KUKA KRL program: MyProgram_339().src

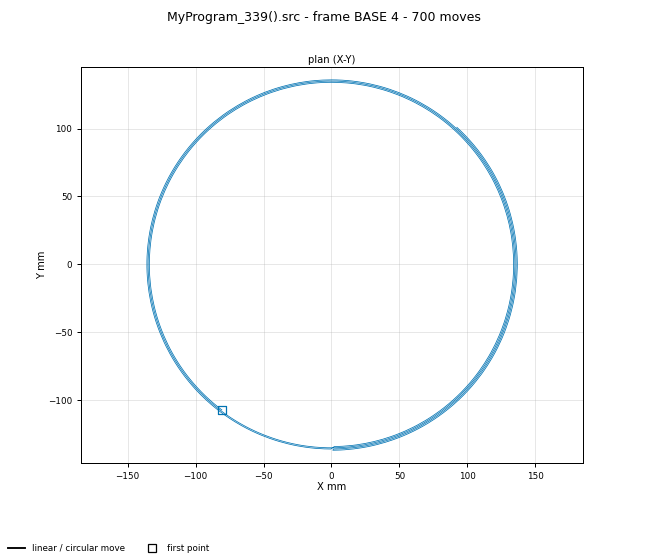
[picture p0: tool path of MyProgram_339().src in frame BASE 4, 700 of 700 moves have a stored position in this frame; points joined in program order, loops and branches not executed]
&ACCESS RVP
&REL 1
&PARAM TEMPLATE = C:\KRC\Roboter\Template\vorgabe
&PARAM EDITMASK = *
DEF MyProgram_339()
; ---- Setting reference (Base) ----
$BASE = BASE_DATA[4]

; --------------------------
; ---- Setting tool (TCP) ----
$TOOL = TOOL_DATA[3]
; --------------------------

$VEL.CP = VEL_APROX_PRINT
Startdeposition()
$VEL.CP = VEL_PRINT
LIN {X -80.6582,Y -106.9926,Z 191,A -116.6087,B 1.012,C 0.191,E1 0.9414,E2 209.5194} C_DIS
LIN {X -83.2208,Y -105.0121,Z 191,A -118.2945,B 1.0123,C 0.1893,E1 0.9375,E2 211.2466} C_DIS
LIN {X -86.7658,Y -102.1022,Z 191,A -120.2784,B 1.0128,C 0.1864,E1 0.9332,E2 213.2337} C_DIS
LIN {X -89.4407,Y -99.7673,Z 191,A -122.0496,B 1.0132,C 0.1842,E1 0.9294,E2 215.0396} C_DIS
LIN {X -92.5437,Y -96.8959,Z 191,A -124.0147,B 1.0137,C 0.1814,E1 0.9254,E2 217.0261} C_DIS
LIN {X -95.7328,Y -93.7464,Z 191,A -126.0613,B 1.0143,C 0.1781,E1 0.9213,E2 219.0903} C_DIS
LIN {X -98.7291,Y -90.5855,Z 191,A -128.1724,B 1.0149,C 0.1749,E1 0.9171,E2 221.2352} C_DIS
LIN {X -101.4585,Y -87.5176,Z 191,A -129.9716,B 1.0154,C 0.1717,E1 0.9138,E2 223.04} C_DIS
LIN {X -103.9869,Y -84.4986,Z 191,A -131.8725,B 1.0159,C 0.1685,E1 0.9103,E2 224.97} C_DIS
LIN {X -106.5269,Y -81.2724,Z 191,A -133.8231,B 1.0165,C 0.165,E1 0.9069,E2 226.9467} C_DIS
LIN {X -108.5873,Y -78.4983,Z 191,A -135.5077,B 1.017,C 0.162,E1 0.9041,E2 228.6589} C_DIS
LIN {X -111.0789,Y -74.9311,Z 191,A -137.5649,B 1.0176,C 0.158,E1 0.9008,E2 230.7422} C_DIS
LIN {X -113.2039,Y -71.6803,Z 191,A -139.4925,B 1.0182,C 0.1544,E1 0.8978,E2 232.7051} C_DIS
LIN {X -115.4642,Y -67.9793,Z 191,A -141.5321,B 1.0188,C 0.1502,E1 0.8948,E2 234.769} C_DIS
LIN {X -117.2157,Y -64.9126,Z 191,A -143.1833,B 1.0193,C 0.1467,E1 0.8925,E2 236.4385} C_DIS
LIN {X -118.7707,Y -62.0179,Z 191,A -144.823,B 1.0198,C 0.1433,E1 0.8903,E2 238.1089} C_DIS
LIN {X -120.4109,Y -58.7718,Z 191,A -146.5306,B 1.0203,C 0.1396,E1 0.8882,E2 239.8362} C_DIS
LIN {X -121.8201,Y -55.7917,Z 191,A -148.1544,B 1.0208,C 0.1361,E1 0.8862,E2 241.4877} C_DIS
LIN {X -123.1512,Y -52.788,Z 191,A -149.9155,B 1.0213,C 0.1325,E1 0.8842,E2 243.2951} C_DIS
LIN {X -124.8857,Y -48.5406,Z 191,A -151.9995,B 1.0219,C 0.1275,E1 0.882,E2 245.3943} C_DIS
LIN {X -126.0829,Y -45.3403,Z 191,A -153.6668,B 1.0224,C 0.1236,E1 0.8804,E2 247.088} C_DIS
LIN {X -127.2363,Y -41.9963,Z 191,A -155.4129,B 1.0228,C 0.1196,E1 0.8788,E2 248.8638} C_DIS
LIN {X -128.2213,Y -38.8855,Z 191,A -156.9641,B 1.0233,C 0.1159,E1 0.8775,E2 250.4347} C_DIS
LIN {X -129.2898,Y -35.1747,Z 191,A -159.129,B 1.0238,C 0.1112,E1 0.8758,E2 252.6651} C_DIS
LIN {X -130.2828,Y -31.2902,Z 191,A -160.9064,B 1.0243,C 0.1065,E1 0.8746,E2 254.4498} C_DIS
LIN {X -131.0111,Y -28.086,Z 191,A -162.5308,B 1.0247,C 0.1026,E1 0.8736,E2 256.1016} C_DIS
LIN {X -131.6609,Y -24.8637,Z 191,A -164.1583,B 1.0251,C 0.0986,E1 0.8727,E2 257.7568} C_DIS
LIN {X -132.289,Y -21.2821,Z 191,A -165.9785,B 1.0255,C 0.0941,E1 0.8719,E2 259.61} C_DIS
LIN {X -132.7236,Y -18.3714,Z 191,A -167.4143,B 1.0258,C 0.0905,E1 0.8713,E2 261.0676} C_DIS
LIN {X -133.1719,Y -14.7703,Z 191,A -169.1065,B 1.0262,C 0.0861,E1 0.8707,E2 262.7767} C_DIS
LIN {X -133.4937,Y -11.4993,Z 191,A -170.8721,B 1.0266,C 0.0819,E1 0.8702,E2 264.5869} C_DIS
LIN {X -133.7359,Y -8.2135,Z 191,A -172.4215,B 1.0269,C 0.0779,E1 0.8699,E2 266.1531} C_DIS
LIN {X -133.8842,Y -5.2709,Z 191,A -173.969,B 1.0271,C 0.0741,E1 0.8697,E2 267.7357} C_DIS
LIN {X -133.9734,Y -1.9867,Z 191,A -175.5899,B 1.0274,C 0.07,E1 0.8697,E2 269.3826} C_DIS
LIN {X -133.9855,Y 0.9522,Z 191,A -177.2293,B 1.0277,C 0.0661,E1 0.8697,E2 271.0686} C_DIS
LIN {X -133.8989,Y 4.8936,Z 191,A -179.0532,B 1.028,C 0.0613,E1 0.8698,E2 272.9085} C_DIS
LIN {X -133.7428,Y 8.102,Z 191,A 179.4246,B 1.0282,C 0.0573,E1 0.87,E2 274.4481} C_DIS
LIN {X -133.5228,Y 11.1541,Z 191,A 177.8434,B 1.0284,C 0.0534,E1 0.8704,E2 276.0618} C_DIS
LIN {X -133.1725,Y 14.7653,Z 191,A 176.0918,B 1.0287,C 0.0489,E1 0.8709,E2 277.8368} C_DIS
LIN {X -132.8155,Y 17.6872,Z 191,A 174.5479,B 1.0288,C 0.0452,E1 0.8714,E2 279.4144} C_DIS
LIN {X -132.3404,Y 20.951,Z 191,A 172.9492,B 1.029,C 0.0411,E1 0.8721,E2 281.035} C_DIS
LIN {X -131.7256,Y 24.525,Z 191,A 171.1308,B 1.0292,C 0.0366,E1 0.873,E2 282.8846} C_DIS
LIN {X -131.0843,Y 27.747,Z 191,A 169.5917,B 1.0292,C 0.0327,E1 0.8739,E2 284.4389} C_DIS
LIN {X -130.4904,Y 30.4188,Z 191,A 167.994,B 1.0294,C 0.0291,E1 0.8749,E2 286.0866} C_DIS
LIN {X -129.5576,Y 34.1706,Z 191,A 166.4075,B 1.0295,C 0.0248,E1 0.876,E2 287.6642} C_DIS
LIN {X -128.6838,Y 37.3263,Z 191,A 164.6242,B 1.0296,C 0.0207,E1 0.8774,E2 289.4919} C_DIS
LIN {X -127.832,Y 40.1504,Z 191,A 163.1708,B 1.0296,C 0.0172,E1 0.8786,E2 290.967} C_DIS
LIN {X -126.699,Y 43.5904,Z 191,A 161.2988,B 1.0297,C 0.0129,E1 0.8803,E2 292.8757} C_DIS
LIN {X -125.2326,Y 47.6435,Z 191,A 159.0965,B 1.0297,C 0.0079,E1 0.8825,E2 295.1186} C_DIS
LIN {X -123.7899,Y 51.2722,Z 191,A 157.5034,B 1.0298,C 0.0038,E1 0.8842,E2 296.7016} C_DIS
LIN {X -122.6365,Y 53.9772,Z 191,A 155.7935,B 1.0298,C 0.0003,E1 0.8861,E2 298.463} C_DIS
LIN {X -121.3505,Y 56.8073,Z 191,A 154.4119,B 1.0298,C -0.003,E1 0.8878,E2 299.8497} C_DIS
LIN {X -119.8894,Y 59.8292,Z 191,A 152.7456,B 1.0298,C -0.0066,E1 0.8898,E2 301.5415} C_DIS
LIN {X -118.166,Y 63.1666,Z 191,A 150.9408,B 1.0298,C -0.0105,E1 0.8922,E2 303.3678} C_DIS
LIN {X -116.5834,Y 66.0427,Z 191,A 149.3435,B 1.0298,C -0.0139,E1 0.8944,E2 304.9862} C_DIS
LIN {X -114.7495,Y 69.1791,Z 191,A 147.4569,B 1.0297,C -0.0176,E1 0.8972,E2 306.9092} C_DIS
LIN {X -112.5008,Y 72.779,Z 191,A 145.4626,B 1.0296,C -0.0217,E1 0.9002,E2 308.9225} C_DIS
LIN {X -110.4885,Y 75.7988,Z 191,A 143.804,B 1.0296,C -0.0251,E1 0.9028,E2 310.592} C_DIS
LIN {X -108.7858,Y 78.2236,Z 191,A 142.3734,B 1.0294,C -0.0279,E1 0.9052,E2 312.0401} C_DIS
LIN {X -106.837,Y 80.8644,Z 191,A 140.9363,B 1.0294,C -0.0308,E1 0.9076,E2 313.48} C_DIS
LIN {X -105.0171,Y 83.2145,Z 191,A 139.2547,B 1.0293,C -0.0334,E1 0.9106,E2 315.2063} C_DIS
LIN {X -102.22,Y 86.6272,Z 191,A 137.1876,B 1.0291,C -0.0372,E1 0.9144,E2 317.2919} C_DIS
LIN {X -99.2737,Y 89.9882,Z 191,A 135.0621,B 1.0291,C -0.0408,E1 0.9184,E2 319.4397} C_DIS
LIN {X -96.4718,Y 92.9862,Z 191,A 133.1168,B 1.0289,C -0.0439,E1 0.9222,E2 321.4046} C_DIS
LIN {X -93.5796,Y 95.8964,Z 191,A 131.3002,B 1.0287,C -0.047,E1 0.9258,E2 323.2269} C_DIS
LIN {X -90.5814,Y 98.7329,Z 191,A 129.2709,B 1.0287,C -0.0498,E1 0.93,E2 325.2836} C_DIS
LIN {X -87.5151,Y 101.4607,Z 191,A 127.5032,B 1.0285,C -0.0526,E1 0.9338,E2 327.0516} C_DIS
LIN {X -84.499,Y 103.9866,Z 191,A 125.6464,B 1.0283,C -0.0551,E1 0.9379,E2 328.9262} C_DIS
LIN {X -81.2745,Y 106.5253,Z 191,A 123.7533,B 1.0283,C -0.0575,E1 0.9421,E2 330.8331} C_DIS
LIN {X -78.9345,Y 108.2711,Z 191,A 122.3198,B 1.0281,C -0.0591,E1 0.9454,E2 332.2857} C_DIS
LIN {X -76.0804,Y 110.2952,Z 191,A 120.8532,B 1.0281,C -0.0611,E1 0.9488,E2 333.7483} C_DIS
LIN {X -73.3552,Y 112.1263,Z 191,A 119.2639,B 1.0279,C -0.0627,E1 0.9526,E2 335.3564} C_DIS
LIN {X -70.57,Y 113.8995,Z 191,A 117.9357,B 1.0279,C -0.0644,E1 0.9557,E2 336.6749} C_DIS
LIN {X -67.7643,Y 115.5905,Z 191,A 116.367,B 1.0277,C -0.0658,E1 0.9596,E2 338.2606} C_DIS
LIN {X -64.918,Y 117.2127,Z 191,A 114.8879,B 1.0277,C -0.0671,E1 0.9632,E2 339.7473} C_DIS
LIN {X -62.0091,Y 118.7753,Z 191,A 113.3972,B 1.0275,C -0.0684,E1 0.967,E2 341.2454} C_DIS
LIN {X -58.7582,Y 120.4177,Z 191,A 111.7712,B 1.0275,C -0.0697,E1 0.9711,E2 342.8778} C_DIS
LIN {X -55.7891,Y 121.8213,Z 191,A 110.3091,B 1.0274,C -0.0708,E1 0.9748,E2 344.3452} C_DIS
LIN {X -52.7868,Y 123.1518,Z 191,A 108.852,B 1.0274,C -0.0718,E1 0.9786,E2 345.8071} C_DIS
LIN {X -50.0675,Y 124.2814,Z 191,A 107.5514,B 1.0273,C -0.0726,E1 0.982,E2 347.1114} C_DIS
LIN {X -47.007,Y 125.471,Z 191,A 106.1033,B 1.0273,C -0.0733,E1 0.9859,E2 348.5633} C_DIS
LIN {X -43.9186,Y 126.5851,Z 191,A 104.6605,B 1.0272,C -0.074,E1 0.9897,E2 350.0095} C_DIS
LIN {X -40.4653,Y 127.7314,Z 191,A 103.0676,B 1.0272,C -0.0747,E1 0.994,E2 351.6055} C_DIS
LIN {X -37.7794,Y 128.5511,Z 191,A 101.8102,B 1.0271,C -0.0751,E1 0.9974,E2 352.8683} C_DIS
LIN {X -34.4694,Y 129.4779,Z 191,A 100.3485,B 1.0271,C -0.0756,E1 1.0014,E2 354.3284} C_DIS
LIN {X -31.2848,Y 130.2841,Z 191,A 98.9263,B 1.0271,C -0.0759,E1 1.0053,E2 355.7517} C_DIS
LIN {X -28.0812,Y 131.0121,Z 191,A 97.51,B 1.027,C -0.0761,E1 1.0092,E2 357.1686} C_DIS
LIN {X -24.8607,Y 131.6614,Z 191,A 96.0961,B 1.027,C -0.0763,E1 1.0131,E2 358.5827} C_DIS
LIN {X -21.2683,Y 132.2912,Z 191,A 94.5183,B 1.027,C -0.0763,E1 1.0175,E2 360.1619} C_DIS
LIN {X -18.3553,Y 132.7259,Z 191,A 93.2012,B 1.027,C -0.0762,E1 1.0212,E2 361.4844} C_DIS
LIN {X -14.7645,Y 133.1725,Z 191,A 91.7254,B 1.027,C -0.0762,E1 1.0254,E2 362.9521} C_DIS
LIN {X -10.5648,Y 133.5726,Z 191,A 89.7687,B 1.027,C -0.0755,E1 1.0309,E2 364.9241} C_DIS
LIN {X -6.9098,Y 133.8097,Z 191,A 88.3975,B 1.027,C -0.0755,E1 1.0347,E2 366.2741} C_DIS
LIN {X -3.616,Y 133.9392,Z 191,A 87.0209,B 1.027,C -0.0751,E1 1.0386,E2 367.6467} C_DIS
LIN {X 0.006,Y 133.99,Z 191,A 85.3856,B 1.0271,C -0.0743,E1 1.0433,E2 369.2905} C_DIS
LIN {X 4.3014,Y 133.9201,Z 191,A 83.5553,B 1.0271,C -0.0734,E1 1.0484,E2 371.1194} C_DIS
LIN {X 8.2243,Y 133.7352,Z 191,A 82.1392,B 1.0272,C -0.0731,E1 1.0523,E2 372.5072} C_DIS
LIN {X 11.1652,Y 133.5219,Z 191,A 80.8463,B 1.0272,C -0.0722,E1 1.056,E2 373.803} C_DIS
LIN {X 14.2409,Y 133.2289,Z 191,A 79.5382,B 1.0273,C -0.0713,E1 1.0597,E2 375.1094} C_DIS
LIN {X 17.6939,Y 132.8146,Z 191,A 78.1152,B 1.0274,C -0.0704,E1 1.0636,E2 376.525} C_DIS
LIN {X 20.9429,Y 132.3416,Z 191,A 76.7975,B 1.0274,C -0.0694,E1 1.0673,E2 377.8332} C_DIS
LIN {X 23.9996,Y 131.8214,Z 191,A 75.4369,B 1.0276,C -0.0682,E1 1.0711,E2 379.1972} C_DIS
LIN {X 27.0615,Y 131.2269,Z 191,A 74.1276,B 1.0276,C -0.067,E1 1.0747,E2 380.5035} C_DIS
LIN {X 30.9581,Y 130.3629,Z 191,A 72.6196,B 1.0277,C -0.0658,E1 1.0788,E2 381.99} C_DIS
LIN {X 34.1462,Y 129.5641,Z 191,A 71.2878,B 1.0277,C -0.0645,E1 1.0824,E2 383.3135} C_DIS
LIN {X 37.3149,Y 128.6871,Z 191,A 70.0343,B 1.0279,C -0.0634,E1 1.0857,E2 384.5503} C_DIS
LIN {X 40.1753,Y 127.824,Z 191,A 68.7562,B 1.0279,C -0.0619,E1 1.0892,E2 385.8283} C_DIS
LIN {X 43.6003,Y 126.6955,Z 191,A 67.4096,B 1.028,C -0.0606,E1 1.0927,E2 387.1536} C_DIS
LIN {X 46.6905,Y 125.5896,Z 191,A 65.9877,B 1.0281,C -0.0587,E1 1.0965,E2 388.5771} C_DIS
LIN {X 49.7536,Y 124.408,Z 191,A 64.7955,B 1.0282,C -0.0575,E1 1.0996,E2 389.7464} C_DIS
LIN {X 52.4719,Y 123.2879,Z 191,A 63.5055,B 1.0283,C -0.0556,E1 1.1029,E2 391.0398} C_DIS
LIN {X 55.7975,Y 121.8175,Z 191,A 62.1712,B 1.0283,C -0.0541,E1 1.1063,E2 392.3499} C_DIS
LIN {X 58.4616,Y 120.5631,Z 191,A 60.8731,B 1.0285,C -0.0521,E1 1.1096,E2 393.6521} C_DIS
LIN {X 61.4387,Y 119.0732,Z 191,A 59.5107,B 1.0285,C -0.05,E1 1.113,E2 395.0077} C_DIS
LIN {X 64.625,Y 117.3749,Z 191,A 58.1389,B 1.0287,C -0.0481,E1 1.1164,E2 396.3605} C_DIS
LIN {X 67.027,Y 116.0196,Z 191,A 56.9624,B 1.0287,C -0.0462,E1 1.1192,E2 397.5366} C_DIS
LIN {X 70.2885,Y 114.0734,Z 191,A 55.5473,B 1.0289,C -0.0442,E1 1.1226,E2 398.9288} C_DIS
LIN {X 72.7712,Y 112.5058,Z 191,A 54.3309,B 1.0289,C -0.0421,E1 1.1255,E2 400.1408} C_DIS
LIN {X 75.8015,Y 110.4866,Z 191,A 53.0372,B 1.029,C -0.0403,E1 1.1284,E2 401.4054} C_DIS
LIN {X 78.2134,Y 108.7931,Z 191,A 51.8101,B 1.0291,C -0.038,E1 1.1312,E2 402.6289} C_DIS
LIN {X 81.1392,Y 106.6287,Z 191,A 50.2799,B 1.0292,C -0.0351,E1 1.1346,E2 404.1561} C_DIS
LIN {X 84.3681,Y 104.0927,Z 191,A 48.6774,B 1.0293,C -0.0323,E1 1.1381,E2 405.7417} C_DIS
LIN {X 87.5177,Y 101.4584,Z 191,A 47.1754,B 1.0293,C -0.0298,E1 1.1413,E2 407.2154} C_DIS
LIN {X 90.5856,Y 98.729,Z 191,A 45.512,B 1.0295,C -0.0265,E1 1.1447,E2 408.8686} C_DIS
LIN {X 93.5678,Y 95.908,Z 191,A 44.0891,B 1.0295,C -0.0243,E1 1.1475,E2 410.2543} C_DIS
LIN {X 95.907,Y 93.5688,Z 191,A 42.7228,B 1.0295,C -0.0214,E1 1.1502,E2 411.6153} C_DIS
LIN {X 98.7283,Y 90.5864,Z 191,A 41.0543,B 1.0297,C -0.0179,E1 1.1534,E2 413.2741} C_DIS
LIN {X 101.4578,Y 87.5184,Z 191,A 39.5878,B 1.0297,C -0.0152,E1 1.156,E2 414.708} C_DIS
LIN {X 103.9847,Y 84.5014,Z 191,A 38.0482,B 1.0297,C -0.012,E1 1.1588,E2 416.2316} C_DIS
LIN {X 106.5303,Y 81.268,Z 191,A 36.4717,B 1.0297,C -0.0087,E1 1.1614,E2 417.7873} C_DIS
LIN {X 109.0106,Y 77.9092,Z 191,A 34.803,B 1.0298,C -0.005,E1 1.1642,E2 419.443} C_DIS
LIN {X 111.2286,Y 74.7095,Z 191,A 33.4156,B 1.0298,C -0.0022,E1 1.1663,E2 420.7988} C_DIS
LIN {X 113.2029,Y 71.6819,Z 191,A 32.0954,B 1.0298,C 0.0005,E1 1.1683,E2 422.0932} C_DIS
LIN {X 114.7477,Y 69.1821,Z 191,A 30.9137,B 1.0298,C 0.0032,E1 1.17,E2 423.2665} C_DIS
LIN {X 116.4141,Y 66.3394,Z 191,A 29.6606,B 1.0298,C 0.006,E1 1.1717,E2 424.5018} C_DIS
LIN {X 118.0059,Y 63.4646,Z 191,A 28.3647,B 1.0298,C 0.0091,E1 1.1734,E2 425.7853} C_DIS
LIN {X 119.6808,Y 60.2453,Z 191,A 27.039,B 1.0298,C 0.0119,E1 1.1751,E2 427.0849} C_DIS
LIN {X 121.1286,Y 57.2779,Z 191,A 25.7774,B 1.0298,C 0.0148,E1 1.1766,E2 428.3292} C_DIS
LIN {X 122.495,Y 54.2937,Z 191,A 24.5348,B 1.0297,C 0.0177,E1 1.178,E2 429.5533} C_DIS
LIN {X 123.7884,Y 51.2759,Z 191,A 23.3318,B 1.0297,C 0.0204,E1 1.1793,E2 430.7329} C_DIS
LIN {X 124.8837,Y 48.5458,Z 191,A 22.1814,B 1.0296,C 0.0232,E1 1.1805,E2 431.8709} C_DIS
LIN {X 126.0021,Y 45.5646,Z 191,A 20.9571,B 1.0295,C 0.0261,E1 1.1816,E2 433.0794} C_DIS
LIN {X 127.1165,Y 42.3561,Z 191,A 19.645,B 1.0294,C 0.0293,E1 1.1828,E2 434.3752} C_DIS
LIN {X 128.2195,Y 38.8913,Z 191,A 18.388,B 1.0294,C 0.032,E1 1.1838,E2 435.5971} C_DIS
LIN {X 129.0434,Y 36.062,Z 191,A 17.2087,B 1.0292,C 0.035,E1 1.1847,E2 436.7672} C_DIS
LIN {X 129.889,Y 32.8865,Z 191,A 15.9691,B 1.0292,C 0.0379,E1 1.1856,E2 437.9873} C_DIS
LIN {X 130.6565,Y 29.6914,Z 191,A 14.8222,B 1.029,C 0.0404,E1 1.1863,E2 439.1035} C_DIS
LIN {X 131.3487,Y 26.4629,Z 191,A 13.4888,B 1.0289,C 0.0439,E1 1.1871,E2 440.4281} C_DIS
LIN {X 131.958,Y 23.2361,Z 191,A 12.2535,B 1.0287,C 0.0469,E1 1.1877,E2 441.6434} C_DIS
LIN {X 132.5396,Y 19.6593,Z 191,A 10.9193,B 1.0286,C 0.0501,E1 1.1882,E2 442.952} C_DIS
LIN {X 132.9808,Y 16.4046,Z 191,A 9.6375,B 1.0284,C 0.0533,E1 1.1887,E2 444.2194} C_DIS
LIN {X 133.3126,Y 13.4502,Z 191,A 8.4422,B 1.0283,C 0.0565,E1 1.189,E2 445.406} C_DIS
LIN {X 133.6253,Y 9.8505,Z 191,A 7.1674,B 1.0281,C 0.0593,E1 1.1893,E2 446.6482} C_DIS
LIN {X 133.8097,Y 6.9111,Z 191,A 6.0568,B 1.0279,C 0.0621,E1 1.1895,E2 447.741} C_DIS
LIN {X 133.9387,Y 3.6313,Z 191,A 4.8744,B 1.0278,C 0.0648,E1 1.1895,E2 448.8967} C_DIS
LIN {X 133.9912,Y -0.0061,Z 191,A 3.4603,B 1.0275,C 0.0684,E1 1.1896,E2 450.2941} C_DIS
LIN {X 133.9531,Y -3.1154,Z 191,A 2.229,B 1.0273,C 0.0716,E1 1.1896,E2 451.5139} C_DIS
LIN {X 133.8264,Y -6.5788,Z 191,A 0.9257,B 1.0271,C 0.0748,E1 1.1894,E2 452.7955} C_DIS
LIN {X 133.5589,Y -10.7268,Z 191,A -0.6786,B 1.0268,C 0.0788,E1 1.1891,E2 454.3792} C_DIS
LIN {X 133.1714,Y -14.7754,Z 191,A -2.0797,B 1.0266,C 0.0818,E1 1.1887,E2 455.7386} C_DIS
LIN {X 132.8137,Y -17.7013,Z 191,A -3.2463,B 1.0263,C 0.0848,E1 1.1883,E2 456.8941} C_DIS
LIN {X 132.3402,Y -20.9518,Z 191,A -4.4561,B 1.0261,C 0.0876,E1 1.1878,E2 458.08} C_DIS
LIN {X 131.7258,Y -24.5243,Z 191,A -5.8362,B 1.0258,C 0.091,E1 1.1871,E2 459.4395} C_DIS
LIN {X 131.0844,Y -27.7465,Z 191,A -7.0727,B 1.0255,C 0.094,E1 1.1864,E2 460.6554} C_DIS
LIN {X 130.4849,Y -30.4427,Z 191,A -8.2143,B 1.0252,C 0.097,E1 1.1857,E2 461.7927} C_DIS
LIN {X 129.5634,Y -34.1489,Z 191,A -9.4872,B 1.025,C 0.0995,E1 1.1849,E2 463.0204} C_DIS
LIN {X 128.6802,Y -37.3385,Z 191,A -10.8022,B 1.0247,C 0.1028,E1 1.1839,E2 464.3234} C_DIS
LIN {X 127.8269,Y -40.1665,Z 191,A -11.9164,B 1.0244,C 0.1055,E1 1.183,E2 465.4193} C_DIS
LIN {X 126.907,Y -42.9854,Z 191,A -13.2309,B 1.024,C 0.1091,E1 1.1818,E2 466.7406} C_DIS
LIN {X 125.2258,Y -47.6617,Z 191,A -15.0452,B 1.0236,C 0.1131,E1 1.1801,E2 468.5162} C_DIS
LIN {X 123.4878,Y -51.9955,Z 191,A -16.74,B 1.0232,C 0.1168,E1 1.1783,E2 470.173} C_DIS
LIN {X 121.8184,Y -55.7953,Z 191,A -18.1521,B 1.0229,C 0.1195,E1 1.1768,E2 471.5389} C_DIS
LIN {X 120.5652,Y -58.4571,Z 191,A -19.3833,B 1.0225,C 0.1226,E1 1.1753,E2 472.7675} C_DIS
LIN {X 119.0909,Y -61.4038,Z 191,A -20.6756,B 1.0221,C 0.1256,E1 1.1737,E2 474.0455} C_DIS
LIN {X 117.5419,Y -64.3202,Z 191,A -21.937,B 1.0218,C 0.1284,E1 1.172,E2 475.2881} C_DIS
LIN {X 115.759,Y -67.4773,Z 191,A -23.2752,B 1.0214,C 0.1312,E1 1.1702,E2 476.5995} C_DIS
LIN {X 114.0709,Y -70.2927,Z 191,A -24.5258,B 1.0211,C 0.1339,E1 1.1684,E2 477.8308} C_DIS
LIN {X 112.4994,Y -72.7811,Z 191,A -25.7065,B 1.0207,C 0.1366,E1 1.1667,E2 479.0021} C_DIS
LIN {X 110.4897,Y -75.797,Z 191,A -27.0414,B 1.0204,C 0.1393,E1 1.1646,E2 480.3096} C_DIS
LIN {X 108.7599,Y -78.2598,Z 191,A -28.1884,B 1.02,C 0.1416,E1 1.1628,E2 481.439} C_DIS
LIN {X 106.6236,Y -81.146,Z 191,A -29.6709,B 1.0196,C 0.145,E1 1.1603,E2 482.9155} C_DIS
LIN {X 104.0974,Y -84.3622,Z 191,A -31.2455,B 1.0191,C 0.1482,E1 1.1576,E2 484.4681} C_DIS
LIN {X 101.4738,Y -87.4999,Z 191,A -32.7292,B 1.0187,C 0.1509,E1 1.1549,E2 485.9175} C_DIS
LIN {X 98.5953,Y -90.731,Z 191,A -34.4639,B 1.0182,C 0.1544,E1 1.1517,E2 487.6381} C_DIS
LIN {X 95.4272,Y -94.058,Z 191,A -36.2368,B 1.0177,C 0.1578,E1 1.1483,E2 489.3867} C_DIS
LIN {X 92.4049,Y -97.0285,Z 191,A -37.8261,B 1.0172,C 0.1606,E1 1.1451,E2 490.9472} C_DIS
LIN {X 89.3326,Y -99.8642,Z 191,A -39.4351,B 1.0168,C 0.1635,E1 1.1419,E2 492.5333} C_DIS
LIN {X 86.2533,Y -102.5356,Z 191,A -41.0206,B 1.0163,C 0.1663,E1 1.1385,E2 494.0988} C_DIS
LIN {X 83.0882,Y -105.1174,Z 191,A -42.7132,B 1.0158,C 0.1695,E1 1.1348,E2 495.7853} C_DIS
LIN {X 79.8038,Y -107.6317,Z 191,A -44.2073,B 1.0154,C 0.1716,E1 1.1316,E2 497.2433} C_DIS
LIN {X 77.1443,Y -109.5533,Z 191,A -45.4196,B 1.0151,C 0.1734,E1 1.1288,E2 498.4306} C_DIS
LIN {X 75.1541,Y -110.928,Z 191,A -46.5151,B 1.0147,C 0.1755,E1 1.1263,E2 499.5351} C_DIS
LIN {X 72.3364,Y -112.7857,Z 191,A -47.8336,B 1.0144,C 0.1776,E1 1.1232,E2 500.8377} C_DIS
LIN {X 69.1842,Y -114.7464,Z 191,A -49.2281,B 1.0141,C 0.1795,E1 1.1199,E2 502.2069} C_DIS
LIN {X 66.3543,Y -116.4056,Z 191,A -50.5262,B 1.0137,C 0.1814,E1 1.1168,E2 503.4916} C_DIS
LIN {X 63.4619,Y -118.0074,Z 191,A -51.8786,B 1.0133,C 0.1834,E1 1.1135,E2 504.8366} C_DIS
LIN {X 60.2432,Y -119.6818,Z 191,A -53.2757,B 1.013,C 0.1853,E1 1.11,E2 506.2136} C_DIS
LIN {X 57.2843,Y -121.1256,Z 191,A -54.5833,B 1.0127,C 0.187,E1 1.1067,E2 507.5083} C_DIS
LIN {X 54.2736,Y -122.504,Z 191,A -55.9017,B 1.0124,C 0.1887,E1 1.1034,E2 508.8142} C_DIS
LIN {X 51.2638,Y -123.7934,Z 191,A -57.2094,B 1.0121,C 0.1903,E1 1.1,E2 510.11} C_DIS
LIN {X 47.5773,Y -125.2574,Z 191,A -58.9331,B 1.0116,C 0.1927,E1 1.0955,E2 511.8388} C_DIS
LIN {X 43.9238,Y -126.5833,Z 191,A -60.3634,B 1.0114,C 0.1939,E1 1.0917,E2 513.2381} C_DIS
LIN {X 40.4641,Y -127.7318,Z 191,A -61.829,B 1.0111,C 0.1955,E1 1.0878,E2 514.6918} C_DIS
LIN {X 37.6457,Y -128.5903,Z 191,A -63.0204,B 1.0109,C 0.1967,E1 1.0846,E2 515.8745} C_DIS
LIN {X 34.4792,Y -129.4753,Z 191,A -64.3549,B 1.0106,C 0.198,E1 1.081,E2 517.2} C_DIS
LIN {X 31.2787,Y -130.2856,Z 191,A -65.6933,B 1.0104,C 0.1992,E1 1.0774,E2 518.5291} C_DIS
LIN {X 28.0766,Y -131.0131,Z 191,A -67.0304,B 1.0101,C 0.2004,E1 1.0737,E2 519.8577} C_DIS
LIN {X 24.8573,Y -131.6621,Z 191,A -68.3708,B 1.0099,C 0.2015,E1 1.07,E2 521.1901} C_DIS
LIN {X 21.2879,Y -132.2881,Z 191,A -69.882,B 1.0097,C 0.2027,E1 1.0659,E2 522.6969} C_DIS
LIN {X 18.3293,Y -132.7296,Z 191,A -71.1606,B 1.0095,C 0.2037,E1 1.0623,E2 523.9762} C_DIS
LIN {X 14.7547,Y -133.1736,Z 191,A -72.481,B 1.0094,C 0.2041,E1 1.0587,E2 525.2669} C_DIS
LIN {X 11.4908,Y -133.4944,Z 191,A -73.9367,B 1.0092,C 0.2053,E1 1.0545,E2 526.7308} C_DIS
LIN {X 8.2177,Y -133.7356,Z 191,A -75.2272,B 1.009,C 0.2058,E1 1.0509,E2 528.0063} C_DIS
LIN {X 5.2603,Y -133.8846,Z 191,A -76.526,B 1.0089,C 0.2066,E1 1.0473,E2 529.3104} C_DIS
LIN {X 1.9832,Y -133.9735,Z 191,A -77.9192,B 1.0087,C 0.2072,E1 1.0433,E2 530.7031} C_DIS
LIN {X 1.9832,Y -133.9735,Z 191,A -77.9192,B 1.0087,C 0.2072,E1 1.0433,E2 530.7031} C_DIS
Enddeposition()
LIN {X 0.9692,Y -134.8761,Z 191,A -78.3976,B 1.0083,C 0.208,E1 1.0416,E2 531.2131} C_DIS
Startdeposition()
$VEL.CP = VEL_PRINT
LIN {X 3.8861,Y -134.8309,Z 191,A -76.0494,B 1.0091,C 0.204,E1 1.0487,E2 528.707} C_DIS
LIN {X 7.9862,Y -134.6505,Z 191,A -74.7012,B 1.0091,C 0.2043,E1 1.0523,E2 527.4141} C_DIS
LIN {X 12.4998,Y -134.3069,Z 191,A -72.8639,B 1.0092,C 0.2033,E1 1.0574,E2 525.5879} C_DIS
LIN {X 19.5941,Y -133.4569,Z 191,A -69.8877,B 1.0097,C 0.2011,E1 1.0658,E2 522.6184} C_DIS
LIN {X 23.3315,Y -132.8542,Z 191,A -68.589,B 1.0097,C 0.2008,E1 1.0693,E2 521.3626} C_DIS
LIN {X 26.7828,Y -132.2009,Z 191,A -67.0718,B 1.01,C 0.1993,E1 1.0735,E2 519.8409} C_DIS
LIN {X 29.4184,Y -131.6409,Z 191,A -65.9962,B 1.0102,C 0.1984,E1 1.0764,E2 518.7743} C_DIS
LIN {X 33.5645,Y -130.6444,Z 191,A -64.0932,B 1.0106,C 0.1962,E1 1.0817,E2 516.8571} C_DIS
LIN {X 37.9879,Y -129.4268,Z 191,A -62.3849,B 1.0109,C 0.1949,E1 1.0862,E2 515.1815} C_DIS
LIN {X 41.2007,Y -128.4402,Z 191,A -61.0271,B 1.0112,C 0.1934,E1 1.0898,E2 513.8326} C_DIS
LIN {X 47.0472,Y -126.4159,Z 191,A -58.5402,B 1.0117,C 0.1906,E1 1.0964,E2 511.3639} C_DIS
LIN {X 49.9749,Y -125.288,Z 191,A -56.5112,B 1.0126,C 0.1859,E1 1.102,E2 509.2354} C_DIS
LIN {X 55.8245,Y -122.795,Z 191,A -54.6444,B 1.0126,C 0.1854,E1 1.1065,E2 507.4848} C_DIS
LIN {X 59.5048,Y -121.0517,Z 191,A -53.2629,B 1.0129,C 0.1843,E1 1.1099,E2 506.151} C_DIS
LIN {X 62.3276,Y -119.6234,Z 191,A -51.9668,B 1.0132,C 0.1823,E1 1.1131,E2 504.8606} C_DIS
LIN {X 65.7431,Y -117.7831,Z 191,A -50.096,B 1.0139,C 0.1787,E1 1.1178,E2 502.9574} C_DIS
LIN {X 68.7585,Y -116.0485,Z 191,A -48.9373,B 1.0141,C 0.1775,E1 1.1205,E2 501.8422} C_DIS
LIN {X 72.429,Y -113.7938,Z 191,A -47.2412,B 1.0145,C 0.1749,E1 1.1245,E2 500.1635} C_DIS
LIN {X 75.5307,Y -111.7586,Z 191,A -45.8537,B 1.0149,C 0.1729,E1 1.1277,E2 498.8011} C_DIS
LIN {X 78.9953,Y -109.3373,Z 191,A -44.3332,B 1.0152,C 0.1708,E1 1.1311,E2 497.3175} C_DIS
LIN {X 81.1046,Y -107.7819,Z 191,A -42.7923,B 1.0159,C 0.1667,E1 1.1347,E2 495.7161} C_DIS
LIN {X 84.5507,Y -105.1002,Z 191,A -40.6748,B 1.0167,C 0.1618,E1 1.1394,E2 493.5605} C_DIS
LIN {X 89.8272,Y -100.6279,Z 191,A -38.9743,B 1.0167,C 0.1617,E1 1.1426,E2 492.0299} C_DIS
LIN {X 94.2566,Y -96.4915,Z 191,A -36.436,B 1.0176,C 0.1564,E1 1.1478,E2 489.4947} C_DIS
LIN {X 100.2456,Y -90.254,Z 191,A -33.3875,B 1.0183,C 0.1514,E1 1.1535,E2 486.5293} C_DIS
LIN {X 104.1335,Y -85.7392,Z 191,A -30.8465,B 1.0192,C 0.1456,E1 1.1581,E2 483.9851} C_DIS
LIN {X 106.1289,Y -83.2557,Z 191,A -28.79,B 1.0201,C 0.1388,E1 1.1618,E2 481.8311} C_DIS
LIN {X 110.5396,Y -77.304,Z 191,A -26.81,B 1.0203,C 0.1373,E1 1.1648,E2 480.0086} C_DIS
LIN {X 113.0595,Y -73.5692,Z 191,A -25.2518,B 1.0207,C 0.1345,E1 1.1671,E2 478.4971} C_DIS
LIN {X 115.0195,Y -70.4654,Z 191,A -23.8529,B 1.0211,C 0.1314,E1 1.1692,E2 477.1186} C_DIS
LIN {X 116.3678,Y -68.2159,Z 191,A -22.7378,B 1.0214,C 0.1286,E1 1.1707,E2 476.0025} C_DIS
LIN {X 118.1133,Y -65.1473,Z 191,A -21.3297,B 1.0219,C 0.1253,E1 1.1726,E2 474.6056} C_DIS
LIN {X 119.9438,Y -61.71,Z 191,A -19.9537,B 1.0222,C 0.1226,E1 1.1744,E2 473.2658} C_DIS
LIN {X 121.6687,Y -58.2328,Z 191,A -18.5699,B 1.0225,C 0.1197,E1 1.176,E2 471.9162} C_DIS
LIN {X 123.4281,Y -54.4091,Z 191,A -16.9704,B 1.0229,C 0.1161,E1 1.1779,E2 470.3405} C_DIS
LIN {X 125.1242,Y -50.3812,Z 191,A -15.2487,B 1.0234,C 0.1119,E1 1.1797,E2 468.6354} C_DIS
LIN {X 126.6091,Y -46.5313,Z 191,A -13.6839,B 1.0238,C 0.1083,E1 1.1812,E2 467.0944} C_DIS
LIN {X 128.1741,Y -42.0253,Z 191,A -11.4285,B 1.0245,C 0.1016,E1 1.1832,E2 464.8072} C_DIS
LIN {X 129.6513,Y -37.2208,Z 191,A -9.9529,B 1.0247,C 0.0994,E1 1.1843,E2 463.4173} C_DIS
LIN {X 130.7363,Y -33.2023,Z 191,A -8.5147,B 1.025,C 0.0963,E1 1.1853,E2 462.0211} C_DIS
LIN {X 131.5613,Y -29.7669,Z 191,A -7.1565,B 1.0253,C 0.093,E1 1.1861,E2 460.6806} C_DIS
LIN {X 132.398,Y -25.7954,Z 191,A -5.7708,B 1.0256,C 0.0901,E1 1.1869,E2 459.3378} C_DIS
LIN {X 132.9777,Y -22.6168,Z 191,A -4.4292,B 1.0259,C 0.0864,E1 1.1875,E2 457.9993} C_DIS
LIN {X 133.5499,Y -18.9437,Z 191,A -3.045,B 1.0261,C 0.0831,E1 1.1881,E2 456.6394} C_DIS
LIN {X 134.0392,Y -15.1124,Z 191,A -1.3623,B 1.0265,C 0.0783,E1 1.1886,E2 454.9503} C_DIS
LIN {X 134.3651,Y -11.8625,Z 191,A -0.3395,B 1.0267,C 0.0765,E1 1.1889,E2 453.9736} C_DIS
LIN {X 134.6012,Y -8.787,Z 191,A 0.81,B 1.0269,C 0.0737,E1 1.1891,E2 452.844} C_DIS
LIN {X 134.773,Y -5.5482,Z 191,A 2.0977,B 1.0271,C 0.0703,E1 1.1893,E2 451.567} C_DIS
LIN {X 134.8852,Y -0.8439,Z 191,A 3.6291,B 1.0273,C 0.0672,E1 1.1893,E2 450.0941} C_DIS
LIN {X 134.851,Y 3.1646,Z 191,A 5.3033,B 1.0276,C 0.0626,E1 1.1893,E2 448.4226} C_DIS
LIN {X 134.7384,Y 6.34,Z 191,A 6.4719,B 1.0278,C 0.0598,E1 1.1891,E2 447.2762} C_DIS
LIN {X 134.4816,Y 10.4666,Z 191,A 7.9073,B 1.0279,C 0.0567,E1 1.1888,E2 445.8804} C_DIS
LIN {X 134.1522,Y 14.0624,Z 191,A 9.3338,B 1.0281,C 0.053,E1 1.1885,E2 444.4665} C_DIS
LIN {X 133.7978,Y 17.1101,Z 191,A 10.4343,B 1.0283,C 0.0504,E1 1.1881,E2 443.3909} C_DIS
LIN {X 133.3039,Y 20.6029,Z 191,A 11.7818,B 1.0284,C 0.0471,E1 1.1875,E2 442.0614} C_DIS
LIN {X 132.6394,Y 24.531,Z 191,A 13.242,B 1.0286,C 0.0436,E1 1.1869,E2 440.6295} C_DIS
LIN {X 131.9169,Y 28.15,Z 191,A 14.6444,B 1.0287,C 0.0402,E1 1.1861,E2 439.2467} C_DIS
LIN {X 131.1117,Y 31.6877,Z 191,A 15.9599,B 1.0288,C 0.0372,E1 1.1853,E2 437.9585} C_DIS
LIN {X 130.3175,Y 34.8098,Z 191,A 17.0735,B 1.0289,C 0.0348,E1 1.1845,E2 436.8756} C_DIS
LIN {X 129.5271,Y 37.6453,Z 191,A 18.3931,B 1.029,C 0.031,E1 1.1835,E2 435.547} C_DIS
LIN {X 128.3641,Y 41.4388,Z 191,A 19.8155,B 1.0291,C 0.0278,E1 1.1823,E2 434.1562} C_DIS
LIN {X 127.0013,Y 45.4434,Z 191,A 21.6157,B 1.0293,C 0.023,E1 1.1806,E2 432.3549} C_DIS
LIN {X 125.2205,Y 50.1423,Z 191,A 23.3111,B 1.0293,C 0.0196,E1 1.179,E2 430.7122} C_DIS
LIN {X 124.125,Y 52.8009,Z 191,A 24.4562,B 1.0293,C 0.0167,E1 1.1777,E2 429.576} C_DIS
LIN {X 122.508,Y 56.446,Z 191,A 26.0274,B 1.0294,C 0.0129,E1 1.1759,E2 428.019} C_DIS
LIN {X 120.3138,Y 60.9831,Z 191,A 27.763,B 1.0294,C 0.0094,E1 1.1738,E2 426.3315} C_DIS
LIN {X 118.638,Y 64.1876,Z 191,A 29.2448,B 1.0294,C 0.0058,E1 1.1719,E2 424.8558} C_DIS
LIN {X 116.7418,Y 67.5737,Z 191,A 30.7114,B 1.0295,C 0.0025,E1 1.1699,E2 423.4106} C_DIS
LIN {X 114.3017,Y 71.6251,Z 191,A 32.4776,B 1.0295,C -0.0013,E1 1.1673,E2 421.6727} C_DIS
LIN {X 112.3292,Y 74.6799,Z 191,A 34.0135,B 1.0295,C -0.005,E1 1.165,E2 420.1375} C_DIS
LIN {X 109.2476,Y 79.1191,Z 191,A 35.8124,B 1.0295,C -0.0082,E1 1.1622,E2 418.3967} C_DIS
LIN {X 106.9082,Y 82.2536,Z 191,A 37.4081,B 1.0295,C -0.0118,E1 1.1595,E2 416.8085} C_DIS
LIN {X 104.1978,Y 85.6611,Z 191,A 39.0304,B 1.0294,C -0.015,E1 1.1567,E2 415.2124} C_DIS
LIN {X 101.5697,Y 88.7607,Z 191,A 40.5616,B 1.0294,C -0.0181,E1 1.1539,E2 413.7036} C_DIS
LIN {X 98.6924,Y 91.9492,Z 191,A 42.2417,B 1.0293,C -0.0215,E1 1.1507,E2 412.04} C_DIS
LIN {X 95.5003,Y 95.2607,Z 191,A 44.0132,B 1.0293,C -0.0249,E1 1.1473,E2 410.2894} C_DIS
LIN {X 92.9733,Y 97.7287,Z 191,A 45.3564,B 1.0291,C -0.0274,E1 1.1446,E2 408.9642} C_DIS
LIN {X 89.6521,Y 100.7845,Z 191,A 47.1128,B 1.0291,C -0.0307,E1 1.141,E2 407.2262} C_DIS
LIN {X 86.3611,Y 103.6185,Z 191,A 48.8048,B 1.029,C -0.0338,E1 1.1374,E2 405.5516} C_DIS
LIN {X 82.8182,Y 106.4709,Z 191,A 50.5537,B 1.0288,C -0.0369,E1 1.1336,E2 403.8235} C_DIS
LIN {X 79.2271,Y 109.1692,Z 191,A 52.3113,B 1.0288,C -0.0399,E1 1.1297,E2 402.083} C_DIS
LIN {X 75.3468,Y 111.8831,Z 191,A 54.0578,B 1.0286,C -0.0425,E1 1.1257,E2 400.3664} C_DIS
LIN {X 71.8466,Y 114.162,Z 191,A 55.7452,B 1.0286,C -0.0454,E1 1.1217,E2 398.6889} C_DIS
LIN {X 68.4599,Y 116.2245,Z 191,A 57.3089,B 1.0284,C -0.0478,E1 1.118,E2 397.1389} C_DIS
LIN {X 65.5029,Y 117.9163,Z 191,A 58.9884,B 1.0282,C -0.0511,E1 1.1138,E2 395.4334} C_DIS
LIN {X 61.8422,Y 119.8765,Z 191,A 60.1826,B 1.0282,C -0.0518,E1 1.111,E2 394.3031} C_DIS
LIN {X 58.5873,Y 121.4993,Z 191,A 61.5131,B 1.0282,C -0.0534,E1 1.1076,E2 392.9965} C_DIS
LIN {X 55.1136,Y 123.113,Z 191,A 63.3238,B 1.028,C -0.0565,E1 1.103,E2 391.1657} C_DIS
LIN {X 50.666,Y 125.0094,Z 191,A 64.8818,B 1.0279,C -0.0576,E1 1.0991,E2 389.6628} C_DIS
LIN {X 47.6671,Y 126.1837,Z 191,A 66.3336,B 1.0278,C -0.0598,E1 1.0952,E2 388.2021} C_DIS
LIN {X 44.8985,Y 127.1968,Z 191,A 67.9928,B 1.0276,C -0.0628,E1 1.0907,E2 386.4983} C_DIS
LIN {X 40.8633,Y 128.548,Z 191,A 69.2325,B 1.0276,C -0.0631,E1 1.0875,E2 385.3215} C_DIS
LIN {X 36.8224,Y 129.7641,Z 191,A 70.9439,B 1.0275,C -0.0649,E1 1.0829,E2 383.6194} C_DIS
LIN {X 33.7147,Y 130.6062,Z 191,A 72.2709,B 1.0274,C -0.0663,E1 1.0793,E2 382.2972} C_DIS
LIN {X 30.1088,Y 131.4833,Z 191,A 73.7879,B 1.0273,C -0.0677,E1 1.0752,E2 380.787} C_DIS
LIN {X 25.6451,Y 132.4267,Z 191,A 75.493,B 1.0273,C -0.0689,E1 1.0705,E2 379.1078} C_DIS
LIN {X 23.0515,Y 132.9043,Z 191,A 76.6047,B 1.0271,C -0.0698,E1 1.0674,E2 377.9974} C_DIS
LIN {X 19.353,Y 133.4914,Z 191,A 78.1541,B 1.0271,C -0.071,E1 1.0631,E2 376.4529} C_DIS
LIN {X 16.4552,Y 133.8801,Z 191,A 79.4239,B 1.027,C -0.0721,E1 1.0595,E2 375.1805} C_DIS
LIN {X 12.7539,Y 134.2825,Z 191,A 80.9159,B 1.027,C -0.0729,E1 1.0554,E2 373.6986} C_DIS
LIN {X 8.482,Y 134.62,Z 191,A 82.691,B 1.0269,C -0.0739,E1 1.0504,E2 371.929} C_DIS
LIN {X 3.9506,Y 134.8291,Z 191,A 84.584,B 1.0268,C -0.0749,E1 1.0451,E2 370.0404} C_DIS
LIN {X -0.3939,Y 134.8868,Z 191,A 86.1443,B 1.0268,C -0.0749,E1 1.0407,E2 368.5114} C_DIS
LIN {X -2.3434,Y 134.8666,Z 191,A 87.3202,B 1.0267,C -0.0761,E1 1.0373,E2 367.2985} C_DIS
LIN {X -7.0055,Y 134.705,Z 191,A 88.9773,B 1.0267,C -0.0761,E1 1.0327,E2 365.6771} C_DIS
LIN {X -10.518,Y 134.4779,Z 191,A 90.727,B 1.0267,C -0.0769,E1 1.0277,E2 363.9007} C_DIS
LIN {X -15.1202,Y 134.0384,Z 191,A 92.6564,B 1.0267,C -0.0771,E1 1.0223,E2 361.9758} C_DIS
LIN {X -18.7559,Y 133.5767,Z 191,A 94.0522,B 1.0267,C -0.0769,E1 1.0185,E2 360.5979} C_DIS
LIN {X -24.4365,Y 132.6564,Z 191,A 96.6363,B 1.0267,C -0.077,E1 1.0112,E2 358.0001} C_DIS
LIN {X -27.8401,Y 131.9838,Z 191,A 97.922,B 1.0267,C -0.0765,E1 1.0077,E2 356.7352} C_DIS
LIN {X -31.2389,Y 131.2199,Z 191,A 99.5134,B 1.0267,C -0.0764,E1 1.0033,E2 355.1325} C_DIS
LIN {X -34.3823,Y 130.4315,Z 191,A 100.9034,B 1.0267,C -0.076,E1 0.9995,E2 353.7418} C_DIS
LIN {X -37.7365,Y 129.5004,Z 191,A 102.4901,B 1.0267,C -0.0756,E1 0.9951,E2 352.1441} C_DIS
LIN {X -42.13,Y 128.1393,Z 191,A 104.6491,B 1.0267,C -0.0751,E1 0.9893,E2 349.9641} C_DIS
LIN {X -46.9998,Y 126.4336,Z 191,A 106.4546,B 1.0269,C -0.0734,E1 0.9846,E2 348.2012} C_DIS
LIN {X -50.3213,Y 125.1483,Z 191,A 107.9234,B 1.0269,C -0.0724,E1 0.9807,E2 346.7379} C_DIS
LIN {X -53.3784,Y 123.8753,Z 191,A 109.4858,B 1.027,C -0.0716,E1 0.9766,E2 345.1596} C_DIS
LIN {X -56.2609,Y 122.5935,Z 191,A 110.9042,B 1.027,C -0.0706,E1 0.973,E2 343.7336} C_DIS
LIN {X -59.7476,Y 120.9319,Z 191,A 112.861,B 1.0272,C -0.0696,E1 0.9679,E2 341.7436} C_DIS
LIN {X -63.8007,Y 118.8458,Z 191,A 114.7014,B 1.0272,C -0.0677,E1 0.9633,E2 339.9147} C_DIS
LIN {X -66.9658,Y 117.0917,Z 191,A 116.564,B 1.0274,C -0.0664,E1 0.9587,E2 338.0177} C_DIS
LIN {X -70.9086,Y 114.7476,Z 191,A 118.9062,B 1.0274,C -0.0645,E1 0.9529,E2 335.6336} C_DIS
LIN {X -73.9878,Y 112.7861,Z 191,A 120.2428,B 1.0276,C -0.0625,E1 0.9498,E2 334.3214} C_DIS
LIN {X -77.3867,Y 110.4822,Z 191,A 122.1644,B 1.0277,C -0.0604,E1 0.9453,E2 332.3814} C_DIS
LIN {X -80.263,Y 108.4105,Z 191,A 123.971,B 1.0278,C -0.0585,E1 0.9411,E2 330.5425} C_DIS
LIN {X -82.9315,Y 106.3831,Z 191,A 125.2972,B 1.028,C -0.0564,E1 0.9382,E2 329.228} C_DIS
LIN {X -86.1439,Y 103.7984,Z 191,A 127.0786,B 1.0281,C -0.0538,E1 0.9343,E2 327.4443} C_DIS
LIN {X -88.9127,Y 101.437,Z 191,A 128.8507,B 1.0282,C -0.0515,E1 0.9305,E2 325.6481} C_DIS
LIN {X -91.4911,Y 99.1176,Z 191,A 130.3917,B 1.0283,C -0.0491,E1 0.9273,E2 324.1005} C_DIS
LIN {X -94.9139,Y 95.845,Z 191,A 132.66,B 1.0285,C -0.0457,E1 0.9227,E2 321.8049} C_DIS
LIN {X -97.8112,Y 92.8871,Z 191,A 134.5832,B 1.0286,C -0.0425,E1 0.9189,E2 319.8644} C_DIS
LIN {X -100.7858,Y 89.6506,Z 191,A 136.7022,B 1.0288,C -0.0391,E1 0.9148,E2 317.7183} C_DIS
LIN {X -103.931,Y 85.9838,Z 191,A 138.8227,B 1.0289,C -0.0351,E1 0.911,E2 315.5913} C_DIS
LIN {X -106.2464,Y 83.1061,Z 191,A 140.5285,B 1.029,C -0.0319,E1 0.908,E2 313.8711} C_DIS
LIN {X -107.9541,Y 80.876,Z 191,A 142.0161,B 1.029,C -0.0294,E1 0.9054,E2 312.351} C_DIS
LIN {X -110.5289,Y 77.3197,Z 191,A 144.0373,B 1.0292,C -0.0254,E1 0.9021,E2 310.313} C_DIS
LIN {X -112.5854,Y 74.2926,Z 191,A 145.7203,B 1.0292,C -0.0219,E1 0.8994,E2 308.6164} C_DIS
LIN {X -114.7271,Y 70.9415,Z 191,A 147.587,B 1.0293,C -0.0181,E1 0.8966,E2 306.7305} C_DIS
LIN {X -116.6709,Y 67.6963,Z 191,A 149.3936,B 1.0294,C -0.0143,E1 0.894,E2 304.9018} C_DIS
LIN {X -118.5673,Y 64.3176,Z 191,A 151.3137,B 1.0294,C -0.0104,E1 0.8914,E2 302.9511} C_DIS
LIN {X -120.0851,Y 61.4325,Z 191,A 152.8618,B 1.0294,C -0.007,E1 0.8893,E2 301.3848} C_DIS
LIN {X -121.5681,Y 58.4433,Z 191,A 154.3252,B 1.0295,C -0.0035,E1 0.8875,E2 299.9169} C_DIS
LIN {X -123.3309,Y 54.6264,Z 191,A 156.6789,B 1.0295,C 0.0013,E1 0.8847,E2 297.4978} C_DIS
LIN {X -124.9004,Y 50.9363,Z 191,A 158.4608,B 1.0295,C 0.0056,E1 0.8828,E2 295.7078} C_DIS
LIN {X -126.2276,Y 47.5499,Z 191,A 160.2876,B 1.0295,C 0.0097,E1 0.8809,E2 293.8486} C_DIS
LIN {X -127.3055,Y 44.5852,Z 191,A 161.7799,B 1.0295,C 0.0133,E1 0.8795,E2 292.339} C_DIS
LIN {X -128.2535,Y 41.785,Z 191,A 163.4324,B 1.0294,C 0.0169,E1 0.878,E2 290.64} C_DIS
LIN {X -129.2573,Y 38.5667,Z 191,A 164.998,B 1.0293,C 0.0208,E1 0.8768,E2 289.0593} C_DIS
LIN {X -130.2936,Y 34.8995,Z 191,A 166.8289,B 1.0292,C 0.0253,E1 0.8754,E2 287.2037} C_DIS
LIN {X -131.9958,Y 27.7845,Z 191,A 170.5002,B 1.0289,C 0.0341,E1 0.873,E2 283.4661} C_DIS
LIN {X -132.7624,Y 23.8441,Z 191,A 172.2125,B 1.0288,C 0.0388,E1 0.8722,E2 281.7538} C_DIS
LIN {X -133.1738,Y 21.4414,Z 191,A 173.5198,B 1.0287,C 0.0419,E1 0.8715,E2 280.414} C_DIS
LIN {X -133.6923,Y 17.9145,Z 191,A 175.265,B 1.0285,C 0.0463,E1 0.8709,E2 278.6413} C_DIS
LIN {X -134.1058,Y 14.4933,Z 191,A 177.0823,B 1.0283,C 0.0506,E1 0.8703,E2 276.7811} C_DIS
LIN {X -134.5137,Y 10.0278,Z 191,A 179.1731,B 1.028,C 0.0561,E1 0.8698,E2 274.6683} C_DIS
LIN {X -134.7073,Y 6.9596,Z 191,A -179.2348,B 1.0278,C 0.06,E1 0.8695,E2 273.0412} C_DIS
LIN {X -134.8567,Y 2.9348,Z 191,A -177.1352,B 1.0274,C 0.0651,E1 0.8693,E2 270.8938} C_DIS
LIN {X -134.8866,Y -0.6335,Z 191,A -175.4626,B 1.0272,C 0.0695,E1 0.8693,E2 269.2023} C_DIS
LIN {X -134.8279,Y -3.9944,Z 191,A -173.7559,B 1.0269,C 0.0737,E1 0.8695,E2 267.461} C_DIS
LIN {X -134.6761,Y -7.5714,Z 191,A -171.9172,B 1.0265,C 0.0782,E1 0.8697,E2 265.5828} C_DIS
LIN {X -134.3985,Y -11.4669,Z 191,A -170.1072,B 1.0262,C 0.083,E1 0.8701,E2 263.7543} C_DIS
LIN {X -134.0221,Y -15.2645,Z 191,A -168.2352,B 1.0258,C 0.0877,E1 0.8707,E2 261.851} C_DIS
LIN {X -133.5828,Y -18.7135,Z 191,A -166.7542,B 1.0254,C 0.0917,E1 0.8712,E2 260.3702} C_DIS
LIN {X -133.083,Y -21.9856,Z 191,A -164.8971,B 1.025,C 0.096,E1 0.8721,E2 258.4556} C_DIS
LIN {X -132.5021,Y -25.2506,Z 191,A -163.2828,B 1.0246,C 0.0999,E1 0.8729,E2 256.8153} C_DIS
LIN {X -131.7981,Y -28.7002,Z 191,A -161.4937,B 1.0242,C 0.1042,E1 0.874,E2 254.9886} C_DIS
LIN {X -130.7977,Y -32.9605,Z 191,A -159.4074,B 1.0237,C 0.1093,E1 0.8753,E2 252.8735} C_DIS
LIN {X -129.6092,Y -37.3647,Z 191,A -157.2043,B 1.0231,C 0.1146,E1 0.877,E2 250.6364} C_DIS
LIN {X -128.6903,Y -40.4175,Z 191,A -155.3124,B 1.0227,C 0.1185,E1 0.8786,E2 248.6741} C_DIS
LIN {X -127.382,Y -44.3643,Z 191,A -153.1408,B 1.0221,C 0.1233,E1 0.8807,E2 246.4492} C_DIS
LIN {X -126.093,Y -47.9092,Z 191,A -151.5565,B 1.0216,C 0.1273,E1 0.8822,E2 244.868} C_DIS
LIN {X -124.7207,Y -51.3761,Z 191,A -149.7961,B 1.0211,C 0.1313,E1 0.8841,E2 243.0845} C_DIS
LIN {X -123.1483,Y -55.0347,Z 191,A -147.9772,B 1.0205,C 0.1356,E1 0.8862,E2 241.2491} C_DIS
LIN {X -121.7758,Y -58.0086,Z 191,A -146.4432,B 1.0201,C 0.139,E1 0.888,E2 239.6964} C_DIS
LIN {X -120.3968,Y -60.8201,Z 191,A -144.9591,B 1.0196,C 0.1422,E1 0.8899,E2 238.192} C_DIS
LIN {X -118.6949,Y -64.0817,Z 191,A -143.0066,B 1.0191,C 0.1459,E1 0.8925,E2 236.1874} C_DIS
LIN {X -116.8642,Y -67.3623,Z 191,A -141.2013,B 1.0186,C 0.1496,E1 0.8951,E2 234.354} C_DIS
LIN {X -114.9049,Y -70.6523,Z 191,A -139.3696,B 1.018,C 0.1533,E1 0.8978,E2 232.4949} C_DIS
LIN {X -112.7725,Y -74.0084,Z 191,A -137.486,B 1.0175,C 0.1569,E1 0.9007,E2 230.5851} C_DIS
LIN {X -110.3056,Y -77.6372,Z 191,A -135.3999,B 1.0169,C 0.1609,E1 0.9041,E2 228.469} C_DIS
LIN {X -107.6754,Y -81.2456,Z 191,A -133.2965,B 1.0162,C 0.1647,E1 0.9077,E2 226.3375} C_DIS
LIN {X -104.9914,Y -84.6857,Z 191,A -131.2598,B 1.0157,C 0.1683,E1 0.9113,E2 224.2758} C_DIS
LIN {X -102.2432,Y -87.984,Z 191,A -129.2664,B 1.0151,C 0.1718,E1 0.9149,E2 222.2592} C_DIS
LIN {X -99.4339,Y -91.1471,Z 191,A -127.4303,B 1.0145,C 0.175,E1 0.9184,E2 220.4179} C_DIS
LIN {X -96.6575,Y -94.0867,Z 191,A -124.6,B 1.0141,C 0.1775,E1 0.9242,E2 217.4327} C_DIS
LIN {X -92.5022,Y -98.1743,Z 191,A -122.3201,B 1.0134,C 0.1817,E1 0.9288,E2 215.1804} C_DIS
LIN {X -89.6544,Y -100.7825,Z 191,A -120.8374,B 1.0129,C 0.1844,E1 0.9319,E2 213.7198} C_DIS
LIN {X -86.2009,Y -103.7511,Z 191,A -118.7701,B 1.0124,C 0.1872,E1 0.9364,E2 211.6339} C_DIS
LIN {X -82.7372,Y -106.5337,Z 191,A -116.7811,B 1.0119,C 0.1897,E1 0.9408,E2 209.6306} C_DIS
LIN {X -79.8072,Y -108.7459,Z 191,A -115.1689,B 1.0115,C 0.1918,E1 0.9445,E2 208.0109} C_DIS
LIN {X -77.658,Y -110.291,Z 191,A -113.8398,B 1.0113,C 0.193,E1 0.9476,E2 206.6529} C_DIS
LIN {X -74.2476,Y -112.6151,Z 191,A -112.0321,B 1.0109,C 0.195,E1 0.9519,E2 204.8374} C_DIS
LIN {X -70.6548,Y -114.9033,Z 191,A -110.1299,B 1.0105,C 0.1969,E1 0.9564,E2 202.9219} C_DIS
LIN {X -67.3275,Y -116.8843,Z 191,A -108.1884,B 1.0102,C 0.1982,E1 0.9613,E2 200.9382} C_DIS
LIN {X -63.16,Y -119.1863,Z 191,A -106.2949,B 1.0098,C 0.2003,E1 0.9659,E2 199.0625} C_DIS
LIN {X -60.0285,Y -120.7934,Z 191,A -104.7239,B 1.0096,C 0.2015,E1 0.9699,E2 197.4805} C_DIS
LIN {X -55.7049,Y -122.8485,Z 191,A -102.6414,B 1.0093,C 0.203,E1 0.9753,E2 195.3906} C_DIS
LIN {X -52.4783,Y -124.2604,Z 191,A -101.0205,B 1.0091,C 0.2038,E1 0.9795,E2 193.7516} C_DIS
LIN {X -49.0435,Y -125.6547,Z 191,A -99.4859,B 1.0089,C 0.2049,E1 0.9835,E2 192.2223} C_DIS
LIN {X -43.8982,Y -127.5437,Z 191,A -97.1144,B 1.0087,C 0.206,E1 0.9899,E2 189.844} C_DIS
LIN {X -40.4789,Y -128.6707,Z 191,A -95.4321,B 1.0087,C 0.2064,E1 0.9944,E2 188.1395} C_DIS
LIN {X -36.7971,Y -129.7712,Z 191,A -93.8183,B 1.0085,C 0.207,E1 0.9988,E2 186.5277} C_DIS
LIN {X -33.0086,Y -130.7854,Z 191,A -92.1508,B 1.0085,C 0.2074,E1 1.0034,E2 184.8593} C_DIS
LIN {X -28.8707,Y -131.7613,Z 191,A -90.2899,B 1.0084,C 0.2076,E1 1.0085,E2 182.9899} C_DIS
LIN {X -25.246,Y -132.503,Z 191,A -88.8443,B 1.0083,C 0.2081,E1 1.0125,E2 181.5616} C_DIS
LIN {X -22.0523,Y -133.0719,Z 191,A -87.3561,B 1.0083,C 0.2079,E1 1.0167,E2 180.0572} C_DIS
LIN {X -18.5409,Y -133.6074,Z 191,A -85.8116,B 1.0083,C 0.2077,E1 1.021,E2 178.5069} C_DIS
LIN {X -15.1101,Y -134.0395,Z 191,A -84.3255,B 1.0083,C 0.2075,E1 1.0252,E2 177.0177} C_DIS
LIN {X -12.158,Y -134.3397,Z 191,A -83.0855,B 1.0084,C 0.2073,E1 1.0287,E2 175.7801} C_DIS
LIN {X -7.3112,Y -134.6896,Z 191,A -81.0093,B 1.0085,C 0.2067,E1 1.0345,E2 173.7011} C_DIS
LIN {X -2.7648,Y -134.8595,Z 191,A -79.3604,B 1.0085,C 0.2069,E1 1.0391,E2 172.0915} C_DIS
LIN {X 0.9692,Y -134.8761,Z 191,A -78.3937,B 1.0083,C 0.2081,E1 1.0416,E2 171.2116} C_DIS
Enddeposition()
LIN {X 0.9692,Y -134.8761,Z 191,A -78.3943,B 1.0083,C 0.2081,E1 1.0416,E2 171.2124} C_DIS
Startdeposition()
$VEL.CP = VEL_PRINT
LIN {X -0.5693,Y -135.7847,Z 191,A -79.4535,B 1.0088,C 0.21,E1 1.0393,E2 172.3552} C_DIS
LIN {X -5.1798,Y -135.687,Z 191,A -80.6484,B 1.0091,C 0.2085,E1 1.0363,E2 173.4445} C_DIS
LIN {X -12.0552,Y -135.2502,Z 191,A -83.7848,B 1.0089,C 0.2099,E1 1.0273,E2 176.6152} C_DIS
LIN {X -15.6631,Y -134.8799,Z 191,A -85.2321,B 1.0089,C 0.2099,E1 1.0233,E2 178.0513} C_DIS
LIN {X -19.3776,Y -134.3959,Z 191,A -86.8477,B 1.0089,C 0.2101,E1 1.0187,E2 179.6726} C_DIS
LIN {X -24.9341,Y -133.4778,Z 191,A -89.0825,B 1.0089,C 0.2097,E1 1.0126,E2 181.8882} C_DIS
LIN {X -27.8316,Y -132.9048,Z 191,A -90.5773,B 1.0089,C 0.2101,E1 1.0083,E2 183.419} C_DIS
LIN {X -31.8549,Y -131.996,Z 191,A -92.2038,B 1.0089,C 0.2095,E1 1.0039,E2 185.0299} C_DIS
LIN {X -35.5281,Y -131.0563,Z 191,A -93.7831,B 1.009,C 0.209,E1 0.9996,E2 186.6069} C_DIS
LIN {X -38.3111,Y -130.2688,Z 191,A -95.064,B 1.0091,C 0.2087,E1 0.9961,E2 187.8968} C_DIS
LIN {X -41.7163,Y -129.2191,Z 191,A -96.5903,B 1.0092,C 0.2081,E1 0.9919,E2 189.4269} C_DIS
LIN {X -45.5068,Y -127.9341,Z 191,A -98.4629,B 1.0093,C 0.2077,E1 0.9869,E2 191.3261} C_DIS
LIN {X -51.7024,Y -125.5586,Z 191,A -101.1473,B 1.0097,C 0.2058,E1 0.9799,E2 193.9949} C_DIS
LIN {X -54.8701,Y -124.2067,Z 191,A -103.1562,B 1.0097,C 0.2057,E1 0.9745,E2 196.0827} C_DIS
LIN {X -58.3824,Y -122.5934,Z 191,A -104.1519,B 1.0102,C 0.2034,E1 0.9721,E2 196.9889} C_DIS
LIN {X -62.0928,Y -120.7576,Z 191,A -106.3172,B 1.0104,C 0.2025,E1 0.9665,E2 199.2138} C_DIS
LIN {X -66.1617,Y -118.579,Z 191,A -108.391,B 1.0107,C 0.2008,E1 0.9613,E2 201.3059} C_DIS
LIN {X -70.9645,Y -115.7679,Z 191,A -110.8438,B 1.0112,C 0.1985,E1 0.9554,E2 203.7737} C_DIS
LIN {X -74.731,Y -113.3731,Z 191,A -113.2519,B 1.0115,C 0.1969,E1 0.9495,E2 206.2557} C_DIS
LIN {X -78.1638,Y -111.0343,Z 191,A -114.7087,B 1.012,C 0.1944,E1 0.9462,E2 207.6712} C_DIS
LIN {X -81.5694,Y -108.5572,Z 191,A -116.6703,B 1.0124,C 0.1922,E1 0.9417,E2 209.6588} C_DIS
LIN {X -85.1675,Y -105.7576,Z 191,A -118.7086,B 1.0129,C 0.1896,E1 0.9372,E2 211.7131} C_DIS
LIN {X -88.619,Y -102.8826,Z 191,A -120.7314,B 1.0134,C 0.1868,E1 0.9328,E2 213.7537} C_DIS
LIN {X -91.8686,Y -99.9917,Z 191,A -122.6201,B 1.0139,C 0.184,E1 0.9288,E2 215.6499} C_DIS
LIN {X -96.2208,Y -95.811,Z 191,A -125.1396,B 1.0147,C 0.1797,E1 0.9237,E2 218.1655} C_DIS
LIN {X -99.6469,Y -92.243,Z 191,A -127.6971,B 1.0153,C 0.1763,E1 0.9186,E2 220.7882} C_DIS
LIN {X -102.1552,Y -89.457,Z 191,A -129.5805,B 1.0158,C 0.1734,E1 0.915,E2 222.713} C_DIS
LIN {X -105.0984,Y -85.9797,Z 191,A -131.694,B 1.0164,C 0.1698,E1 0.9112,E2 224.8526} C_DIS
LIN {X -107.7327,Y -82.6551,Z 191,A -133.5891,B 1.017,C 0.1663,E1 0.9079,E2 226.7619} C_DIS
LIN {X -110.1675,Y -79.3815,Z 191,A -135.63,B 1.0175,C 0.1628,E1 0.9044,E2 228.8462} C_DIS
LIN {X -112.7574,Y -75.6574,Z 191,A -137.776,B 1.0182,C 0.1587,E1 0.901,E2 231.0234} C_DIS
LIN {X -114.9669,Y -72.2555,Z 191,A -139.5775,B 1.0188,C 0.1549,E1 0.8982,E2 232.8367} C_DIS
LIN {X -116.7836,Y -69.2809,Z 191,A -141.2647,B 1.0192,C 0.1516,E1 0.8958,E2 234.5529} C_DIS
LIN {X -118.6213,Y -66.0855,Z 191,A -143.4661,B 1.0198,C 0.1479,E1 0.8926,E2 236.841} C_DIS
LIN {X -120.4655,Y -62.6575,Z 191,A -144.81,B 1.0203,C 0.1442,E1 0.8909,E2 238.1443} C_DIS
LIN {X -121.8847,Y -59.8482,Z 191,A -146.3592,B 1.0208,C 0.1409,E1 0.889,E2 239.7228} C_DIS
LIN {X -123.396,Y -56.6673,Z 191,A -147.9994,B 1.0213,C 0.1373,E1 0.887,E2 241.3831} C_DIS
LIN {X -124.7244,Y -53.6796,Z 191,A -149.5897,B 1.0217,C 0.1338,E1 0.8852,E2 243.0011} C_DIS
LIN {X -126.0113,Y -50.5848,Z 191,A -151.2244,B 1.0222,C 0.1302,E1 0.8834,E2 244.6646} C_DIS
LIN {X -127.5683,Y -46.5213,Z 191,A -153.5774,B 1.0228,C 0.1252,E1 0.881,E2 247.0855} C_DIS
LIN {X -129.0546,Y -42.2263,Z 191,A -155.5325,B 1.0234,C 0.1203,E1 0.8793,E2 249.0448} C_DIS
LIN {X -130.1829,Y -38.6044,Z 191,A -157.4554,B 1.0239,C 0.1159,E1 0.8777,E2 251.0094} C_DIS
LIN {X -131.2941,Y -34.6361,Z 191,A -159.375,B 1.0245,C 0.1112,E1 0.8762,E2 252.9519} C_DIS
LIN {X -132.066,Y -31.5648,Z 191,A -161.0278,B 1.0249,C 0.1074,E1 0.8751,E2 254.6453} C_DIS
LIN {X -133.0117,Y -27.3064,Z 191,A -163.0652,B 1.0254,C 0.1023,E1 0.8739,E2 256.7074} C_DIS
LIN {X -133.7011,Y -23.702,Z 191,A -164.8384,B 1.0258,C 0.0979,E1 0.873,E2 258.5089} C_DIS
LIN {X -134.1989,Y -20.6977,Z 191,A -166.3348,B 1.0262,C 0.0942,E1 0.8723,E2 260.032} C_DIS
LIN {X -134.6699,Y -17.3729,Z 191,A -167.9295,B 1.0265,C 0.0901,E1 0.8717,E2 261.6488} C_DIS
LIN {X -135.0284,Y -14.3215,Z 191,A -169.5847,B 1.0268,C 0.0863,E1 0.8712,E2 263.3492} C_DIS
LIN {X -135.4187,Y -9.977,Z 191,A -171.635,B 1.0273,C 0.081,E1 0.8707,E2 265.4252} C_DIS
LIN {X -135.6547,Y -6.0068,Z 191,A -173.746,B 1.0277,C 0.0759,E1 0.8704,E2 267.5902} C_DIS
LIN {X -135.7726,Y -1.9214,Z 191,A -175.6921,B 1.028,C 0.0709,E1 0.8703,E2 269.5632} C_DIS
LIN {X -135.7616,Y 2.5845,Z 191,A -177.7786,B 1.0284,C 0.0654,E1 0.8703,E2 271.6718} C_DIS
LIN {X -135.6603,Y 5.8639,Z 191,A -179.5691,B 1.0286,C 0.0612,E1 0.8705,E2 273.5122} C_DIS
LIN {X -135.4197,Y 9.9637,Z 191,A 178.538,B 1.0289,C 0.0562,E1 0.8709,E2 275.4239} C_DIS
LIN {X -135.13,Y 13.3326,Z 191,A 176.7994,B 1.0292,C 0.052,E1 0.8713,E2 277.2002} C_DIS
LIN {X -134.6539,Y 17.4953,Z 191,A 174.8353,B 1.0294,C 0.0469,E1 0.872,E2 279.1873} C_DIS
LIN {X -134.1842,Y 20.7926,Z 191,A 173.1847,B 1.0296,C 0.0428,E1 0.8727,E2 280.8671} C_DIS
LIN {X -133.5685,Y 24.443,Z 191,A 171.4483,B 1.0297,C 0.0384,E1 0.8735,E2 282.6239} C_DIS
LIN {X -132.9074,Y 27.8191,Z 191,A 169.5451,B 1.0299,C 0.034,E1 0.8746,E2 284.5809} C_DIS
LIN {X -131.6667,Y 33.1904,Z 191,A 167.032,B 1.0301,C 0.0276,E1 0.8763,E2 287.1151} C_DIS
LIN {X -130.7779,Y 36.535,Z 191,A 165.3176,B 1.0301,C 0.0235,E1 0.8776,E2 288.859} C_DIS
LIN {X -129.877,Y 39.6189,Z 191,A 163.7214,B 1.0303,C 0.0197,E1 0.8789,E2 290.4831} C_DIS
LIN {X -128.7381,Y 43.1768,Z 191,A 161.9729,B 1.0303,C 0.0155,E1 0.8804,E2 292.2511} C_DIS
LIN {X -127.6323,Y 46.3436,Z 191,A 160.3504,B 1.0303,C 0.0117,E1 0.8819,E2 293.8972} C_DIS
LIN {X -126.4027,Y 49.6002,Z 191,A 158.6289,B 1.0304,C 0.0077,E1 0.8837,E2 295.6475} C_DIS
LIN {X -124.8068,Y 53.4892,Z 191,A 156.4481,B 1.0304,C 0.003,E1 0.8861,E2 297.8748} C_DIS
LIN {X -123.1948,Y 57.1023,Z 191,A 154.7685,B 1.0304,C -0.0011,E1 0.8881,E2 299.5545} C_DIS
LIN {X -121.7752,Y 60.0702,Z 191,A 153.1484,B 1.0304,C -0.0046,E1 0.8901,E2 301.2007} C_DIS
LIN {X -119.6701,Y 64.1658,Z 191,A 150.8268,B 1.0304,C -0.0094,E1 0.8931,E2 303.5648} C_DIS
LIN {X -117.5999,Y 67.8857,Z 191,A 148.5886,B 1.0304,C -0.0138,E1 0.8963,E2 305.8526} C_DIS
LIN {X -115.3813,Y 71.5916,Z 191,A 146.7256,B 1.0304,C -0.018,E1 0.899,E2 307.7189} C_DIS
LIN {X -112.9098,Y 75.429,Z 191,A 144.5846,B 1.0302,C -0.0223,E1 0.9024,E2 309.8832} C_DIS
LIN {X -110.4773,Y 78.9489,Z 191,A 142.4779,B 1.0302,C -0.0262,E1 0.9058,E2 312.0228} C_DIS
LIN {X -107.9754,Y 82.3378,Z 191,A 140.5208,B 1.03,C -0.0299,E1 0.9092,E2 313.999} C_DIS
LIN {X -105.1562,Y 85.9089,Z 191,A 138.0708,B 1.03,C -0.0338,E1 0.9136,E2 316.5068} C_DIS
LIN {X -102.704,Y 88.8264,Z 191,A 136.0984,B 1.0298,C -0.0369,E1 0.9173,E2 318.5185} C_DIS
LIN {X -99.5699,Y 92.326,Z 191,A 134.7829,B 1.0297,C -0.0406,E1 0.9196,E2 319.7589} C_DIS
LIN {X -96.0578,Y 95.975,Z 191,A 131.6309,B 1.0295,C -0.0443,E1 0.9261,E2 323.0217} C_DIS
LIN {X -92.891,Y 99.0434,Z 191,A 129.8459,B 1.0294,C -0.0474,E1 0.9297,E2 324.7972} C_DIS
LIN {X -89.3162,Y 102.278,Z 191,A 127.8405,B 1.0292,C -0.0507,E1 0.9339,E2 326.7982} C_DIS
LIN {X -86.096,Y 105.0033,Z 191,A 125.9459,B 1.0291,C -0.0533,E1 0.938,E2 328.7042} C_DIS
LIN {X -79.6837,Y 109.9485,Z 191,A 122.5747,B 1.0288,C -0.0581,E1 0.9456,E2 332.0685} C_DIS
LIN {X -75.7482,Y 112.6968,Z 191,A 120.1512,B 1.0287,C -0.0605,E1 0.9513,E2 334.5342} C_DIS
LIN {X -69.1734,Y 116.8477,Z 191,A 116.0975,B 1.0285,C -0.0636,E1 0.9612,E2 338.6689} C_DIS
LIN {X -65.1358,Y 119.1449,Z 191,A 114.8954,B 1.0283,C -0.0662,E1 0.964,E2 339.7886} C_DIS
LIN {X -62.9089,Y 120.3335,Z 191,A 113.487,B 1.0283,C -0.067,E1 0.9676,E2 341.2333} C_DIS
LIN {X -59.0602,Y 122.2696,Z 191,A 111.3976,B 1.0283,C -0.0683,E1 0.9729,E2 343.3509} C_DIS
LIN {X -54.8654,Y 124.2087,Z 191,A 109.6049,B 1.0281,C -0.0699,E1 0.9775,E2 345.1257} C_DIS
LIN {X -51.8085,Y 125.5143,Z 191,A 108.1534,B 1.0281,C -0.0709,E1 0.9813,E2 346.5816} C_DIS
LIN {X -48.5145,Y 126.8248,Z 191,A 106.6022,B 1.028,C -0.0717,E1 0.9854,E2 348.138} C_DIS
LIN {X -42.5897,Y 128.9336,Z 191,A 103.8807,B 1.0279,C -0.073,E1 0.9927,E2 350.8653} C_DIS
LIN {X -39.5699,Y 129.8919,Z 191,A 102.4797,B 1.0279,C -0.0735,E1 0.9965,E2 352.2726} C_DIS
LIN {X -36.0644,Y 130.9096,Z 191,A 100.936,B 1.0279,C -0.074,E1 1.0007,E2 353.8158} C_DIS
LIN {X -32.9531,Y 131.727,Z 191,A 99.6003,B 1.0278,C -0.0744,E1 1.0043,E2 355.1487} C_DIS
LIN {X -29.9538,Y 132.4407,Z 191,A 98.2949,B 1.0278,C -0.0747,E1 1.0079,E2 356.4539} C_DIS
LIN {X -27.119,Y 133.0499,Z 191,A 97,B 1.0278,C -0.0747,E1 1.0115,E2 357.7558} C_DIS
LIN {X -23.7036,Y 133.7008,Z 191,A 95.2946,B 1.0278,C -0.0744,E1 1.0163,E2 359.4859} C_DIS
LIN {X -18.0891,Y 134.5761,Z 191,A 93.2113,B 1.0278,C -0.075,E1 1.022,E2 361.5347} C_DIS
LIN {X -15.1127,Y 134.9433,Z 191,A 91.8031,B 1.0278,C -0.0746,E1 1.026,E2 362.9576} C_DIS
LIN {X -11.1726,Y 135.3255,Z 191,A 89.637,B 1.0278,C -0.0732,E1 1.0323,E2 365.1753} C_DIS
LIN {X -6.3751,Y 135.6367,Z 191,A 88.2414,B 1.0278,C -0.0741,E1 1.036,E2 366.5032} C_DIS
LIN {X 0.1059,Y 135.7873,Z 191,A 85.6065,B 1.0278,C -0.0732,E1 1.0435,E2 369.1264} C_DIS
LIN {X 3.5998,Y 135.7382,Z 191,A 83.5787,B 1.028,C -0.0712,E1 1.0493,E2 371.2124} C_DIS
LIN {X 8.0648,Y 135.5463,Z 191,A 81.9138,B 1.028,C -0.0706,E1 1.054,E2 372.8533} C_DIS
LIN {X 11.5903,Y 135.2902,Z 191,A 80.7926,B 1.028,C -0.0706,E1 1.057,E2 373.9345} C_DIS
LIN {X 15.1437,Y 134.94,Z 191,A 79.2748,B 1.0281,C -0.0696,E1 1.0613,E2 375.453} C_DIS
LIN {X 19.4119,Y 134.391,Z 191,A 77.3494,B 1.0282,C -0.0678,E1 1.0667,E2 377.3895} C_DIS
LIN {X 24.455,Y 133.5663,Z 191,A 75.4102,B 1.0283,C -0.0665,E1 1.072,E2 379.3049} C_DIS
LIN {X 28.5956,Y 132.7403,Z 191,A 73.8276,B 1.0283,C -0.0654,E1 1.0763,E2 380.8655} C_DIS
LIN {X 32.3922,Y 131.8665,Z 191,A 72.3002,B 1.0285,C -0.0641,E1 1.0805,E2 382.38} C_DIS
LIN {X 34.9843,Y 131.2013,Z 191,A 71.1814,B 1.0285,C -0.0629,E1 1.0835,E2 383.4973} C_DIS
LIN {X 38.7314,Y 130.1457,Z 191,A 69.6559,B 1.0286,C -0.0614,E1 1.0876,E2 385.0098} C_DIS
LIN {X 42.5563,Y 128.9448,Z 191,A 67.9921,B 1.0288,C -0.0594,E1 1.0921,E2 386.6702} C_DIS
LIN {X 49.6144,Y 126.3972,Z 191,A 65.0092,B 1.029,C -0.0558,E1 1.0999,E2 389.6324} C_DIS
LIN {X 55.6955,Y 123.8375,Z 191,A 62.4635,B 1.0291,C -0.0527,E1 1.1065,E2 392.1517} C_DIS
LIN {X 58.7129,Y 122.4355,Z 191,A 61.2025,B 1.0291,C -0.0511,E1 1.1096,E2 393.3967} C_DIS
LIN {X 61.7821,Y 120.9158,Z 191,A 59.8615,B 1.0293,C -0.0492,E1 1.113,E2 394.726} C_DIS
LIN {X 64.8886,Y 119.2798,Z 191,A 57.613,B 1.0295,C -0.0438,E1 1.1188,E2 397.0585} C_DIS
LIN {X 70.6694,Y 115.949,Z 191,A 55.3743,B 1.0296,C -0.0412,E1 1.124,E2 399.234} C_DIS
LIN {X 74.5423,Y 113.4973,Z 191,A 54.3435,B 1.0296,C -0.0413,E1 1.1262,E2 400.1644} C_DIS
LIN {X 78.6738,Y 110.6741,Z 191,A 52.043,B 1.0298,C -0.0366,E1 1.1315,E2 402.4859} C_DIS
LIN {X 82.3306,Y 107.9809,Z 191,A 50.3229,B 1.0299,C -0.0338,E1 1.1354,E2 404.1841} C_DIS
LIN {X 85.5907,Y 105.4163,Z 191,A 48.7213,B 1.03,C -0.0309,E1 1.1388,E2 405.7689} C_DIS
LIN {X 89.0238,Y 102.5331,Z 191,A 46.9866,B 1.03,C -0.0277,E1 1.1425,E2 407.4859} C_DIS
LIN {X 92.3923,Y 99.5081,Z 191,A 45.4621,B 1.0302,C -0.0254,E1 1.1456,E2 408.9667} C_DIS
LIN {X 94.8042,Y 97.2135,Z 191,A 43.9891,B 1.0302,C -0.0221,E1 1.1486,E2 410.4476} C_DIS
LIN {X 98.0068,Y 93.9834,Z 191,A 42.2885,B 1.0302,C -0.0189,E1 1.1519,E2 412.1233} C_DIS
LIN {X 100.9069,Y 90.8631,Z 191,A 40.6868,B 1.0303,C -0.0158,E1 1.1549,E2 413.7027} C_DIS
LIN {X 103.7165,Y 87.6426,Z 191,A 39.0323,B 1.0303,C -0.0123,E1 1.1578,E2 415.3403} C_DIS
LIN {X 106.5399,Y 84.1878,Z 191,A 37.3721,B 1.0304,C -0.009,E1 1.1607,E2 416.975} C_DIS
LIN {X 109.2001,Y 80.7072,Z 191,A 35.6669,B 1.0304,C -0.0053,E1 1.1636,E2 418.6639} C_DIS
LIN {X 111.8531,Y 76.9876,Z 191,A 33.4389,B 1.0304,C 0.0009,E1 1.1672,E2 420.9271} C_DIS
LIN {X 114.8436,Y 72.4508,Z 191,A 32.1377,B 1.0304,C 0.0017,E1 1.169,E2 422.113} C_DIS
LIN {X 117.7187,Y 67.6805,Z 191,A 29.932,B 1.0304,C 0.0069,E1 1.1721,E2 424.3022} C_DIS
LIN {X 119.5177,Y 64.4494,Z 191,A 28.4582,B 1.0304,C 0.0104,E1 1.1741,E2 425.7661} C_DIS
LIN {X 121.3321,Y 60.9644,Z 191,A 27.0653,B 1.0304,C 0.0133,E1 1.1758,E2 427.1279} C_DIS
LIN {X 122.5917,Y 58.386,Z 191,A 25.5306,B 1.0304,C 0.0181,E1 1.1777,E2 428.7015} C_DIS
LIN {X 124.4631,Y 54.2839,Z 191,A 24.4382,B 1.0303,C 0.019,E1 1.1789,E2 429.6977} C_DIS
LIN {X 125.7359,Y 51.2681,Z 191,A 22.4919,B 1.0301,C 0.0255,E1 1.181,E2 431.7122} C_DIS
LIN {X 127.6174,Y 46.3852,Z 191,A 21.2872,B 1.0301,C 0.0263,E1 1.182,E2 432.7969} C_DIS
LIN {X 128.8192,Y 42.9333,Z 191,A 19.728,B 1.0301,C 0.0305,E1 1.1834,E2 434.3587} C_DIS
LIN {X 129.9686,Y 39.3193,Z 191,A 18.245,B 1.0299,C 0.0342,E1 1.1847,E2 435.8281} C_DIS
LIN {X 131.1595,Y 35.141,Z 191,A 16.7326,B 1.0298,C 0.0375,E1 1.1858,E2 437.3019} C_DIS
LIN {X 131.99,Y 31.8798,Z 191,A 15.451,B 1.0297,C 0.0407,E1 1.1866,E2 438.5672} C_DIS
LIN {X 132.822,Y 28.2171,Z 191,A 14.0608,B 1.0295,C 0.044,E1 1.1874,E2 439.9341} C_DIS
LIN {X 133.8018,Y 23.1388,Z 191,A 12.0604,B 1.0293,C 0.0491,E1 1.1884,E2 441.913} C_DIS
LIN {X 134.4623,Y 18.9129,Z 191,A 10.5521,B 1.0291,C 0.0525,E1 1.189,E2 443.3853} C_DIS
LIN {X 135.127,Y 13.3634,Z 191,A 7.9628,B 1.0287,C 0.0603,E1 1.1898,E2 446.0045} C_DIS
LIN {X 135.5211,Y 8.4739,Z 191,A 6.9017,B 1.0287,C 0.0607,E1 1.19,E2 446.9404} C_DIS
LIN {X 135.7263,Y 4.0281,Z 191,A 4.4664,B 1.0282,C 0.0689,E1 1.1903,E2 449.4468} C_DIS
LIN {X 135.7825,Y -1.0774,Z 191,A 3.1244,B 1.028,C 0.0706,E1 1.1903,E2 450.6877} C_DIS
LIN {X 135.5679,Y -7.7151,Z 191,A 0.7184,B 1.0276,C 0.0763,E1 1.19,E2 453.0449} C_DIS
LIN {X 135.3447,Y -10.9455,Z 191,A -1.2657,B 1.0271,C 0.0834,E1 1.1896,E2 455.1084} C_DIS
LIN {X 134.7155,Y -17.025,Z 191,A -2.7527,B 1.027,C 0.0847,E1 1.1891,E2 456.4575} C_DIS
LIN {X 134.2257,Y -20.5242,Z 191,A -4.1779,B 1.0267,C 0.0884,E1 1.1885,E2 457.8751} C_DIS
LIN {X 133.6148,Y -24.1842,Z 191,A -5.5437,B 1.0264,C 0.0917,E1 1.1879,E2 459.2161} C_DIS
LIN {X 132.7775,Y -28.4233,Z 191,A -7.1819,B 1.026,C 0.0957,E1 1.187,E2 460.8314} C_DIS
LIN {X 131.9417,Y -32.0804,Z 191,A -8.5076,B 1.0257,C 0.0986,E1 1.1862,E2 462.1247} C_DIS
LIN {X 131.1723,Y -35.093,Z 191,A -9.727,B 1.0254,C 0.1017,E1 1.1853,E2 463.3328} C_DIS
LIN {X 130.1616,Y -38.6773,Z 191,A -11.0823,B 1.0251,C 0.1048,E1 1.1843,E2 464.6609} C_DIS
LIN {X 127.4119,Y -46.9507,Z 191,A -14.3824,B 1.0243,C 0.1127,E1 1.1814,E2 467.9138} C_DIS
LIN {X 124.5675,Y -54.0426,Z 191,A -17.1988,B 1.0236,C 0.119,E1 1.1784,E2 470.6785} C_DIS
LIN {X 123.0915,Y -57.3257,Z 191,A -18.5082,B 1.0232,C 0.1218,E1 1.1769,E2 471.9611} C_DIS
LIN {X 121.4926,Y -60.6431,Z 191,A -19.9094,B 1.0229,C 0.125,E1 1.1752,E2 473.3432} C_DIS
LIN {X 119.6944,Y -64.1205,Z 191,A -21.4623,B 1.0224,C 0.1287,E1 1.1732,E2 474.8841} C_DIS
LIN {X 117.6523,Y -67.7951,Z 191,A -23.1653,B 1.0219,C 0.1328,E1 1.1709,E2 476.5789} C_DIS
LIN {X 115.7877,Y -70.9323,Z 191,A -24.4461,B 1.0215,C 0.1353,E1 1.1691,E2 477.8261} C_DIS
LIN {X 113.3798,Y -74.7208,Z 191,A -26.1836,B 1.021,C 0.1391,E1 1.1665,E2 479.5439} C_DIS
LIN {X 110.5961,Y -78.7828,Z 191,A -28.0297,B 1.0205,C 0.1429,E1 1.1636,E2 481.3603} C_DIS
LIN {X 106.1972,Y -84.6187,Z 191,A -30.3919,B 1.02,C 0.1465,E1 1.1597,E2 483.6267} C_DIS
LIN {X 101.8632,Y -89.7892,Z 191,A -33.3282,B 1.019,C 0.1535,E1 1.1544,E2 486.5774} C_DIS
LIN {X 97.0582,Y -94.9626,Z 191,A -35.7034,B 1.0184,C 0.1571,E1 1.15,E2 488.8721} C_DIS
LIN {X 94.9795,Y -97.0416,Z 191,A -37.1048,B 1.0179,C 0.1605,E1 1.1471,E2 490.2967} C_DIS
LIN {X 91.8425,Y -100.0157,Z 191,A -38.8529,B 1.0173,C 0.164,E1 1.1436,E2 492.0357} C_DIS
LIN {X 85.9898,Y -105.0901,Z 191,A -41.7332,B 1.0166,C 0.1688,E1 1.1375,E2 494.8649} C_DIS
LIN {X 82.5817,Y -107.7889,Z 191,A -43.697,B 1.0159,C 0.1729,E1 1.1331,E2 496.848} C_DIS
LIN {X 79.4637,Y -110.108,Z 191,A -44.9644,B 1.0156,C 0.1743,E1 1.1303,E2 498.0652} C_DIS
LIN {X 76.434,Y -112.2326,Z 191,A -46.3893,B 1.0152,C 0.1766,E1 1.1271,E2 499.4723} C_DIS
LIN {X 72.7165,Y -114.6759,Z 191,A -48.0401,B 1.0148,C 0.1789,E1 1.1232,E2 501.093} C_DIS
LIN {X 65.8598,Y -118.7462,Z 191,A -51.0317,B 1.0141,C 0.183,E1 1.1161,E2 504.035} C_DIS
LIN {X 62.647,Y -120.471,Z 191,A -52.5217,B 1.0137,C 0.1853,E1 1.1124,E2 505.5193} C_DIS
LIN {X 59.5228,Y -122.0452,Z 191,A -53.8957,B 1.0133,C 0.1871,E1 1.109,E2 506.8801} C_DIS
LIN {X 55.8536,Y -123.7667,Z 191,A -56.338,B 1.0123,C 0.1927,E1 1.1025,E2 509.4259} C_DIS
LIN {X 49.7064,Y -126.3615,Z 191,A -58.0232,B 1.0124,C 0.192,E1 1.0985,E2 510.9549} C_DIS
LIN {X 47.1537,Y -127.3359,Z 191,A -59.3725,B 1.012,C 0.1943,E1 1.0948,E2 512.3327} C_DIS
LIN {X 42.6643,Y -128.9088,Z 191,A -61.0859,B 1.0117,C 0.1957,E1 1.0903,E2 514.006} C_DIS
LIN {X 39.4449,Y -129.9302,Z 191,A -62.4353,B 1.0114,C 0.1971,E1 1.0867,E2 515.3457} C_DIS
LIN {X 36.5018,Y -130.7872,Z 191,A -63.694,B 1.0112,C 0.1985,E1 1.0833,E2 516.6003} C_DIS
LIN {X 33.1294,Y -131.6822,Z 191,A -65.0769,B 1.0109,C 0.1997,E1 1.0796,E2 517.9716} C_DIS
LIN {X 29.1152,Y -132.6281,Z 191,A -66.5875,B 1.0107,C 0.2007,E1 1.0755,E2 519.4507} C_DIS
LIN {X 24.2921,Y -133.5955,Z 191,A -68.7619,B 1.0103,C 0.203,E1 1.0695,E2 521.6405} C_DIS
LIN {X 17.9578,Y -134.5933,Z 191,A -71.3867,B 1.0099,C 0.2049,E1 1.0622,E2 524.2555} C_DIS
LIN {X 9.3828,Y -135.4621,Z 191,A -74.8053,B 1.0095,C 0.2067,E1 1.0526,E2 527.6453} C_DIS
LIN {X 1.4759,Y -135.7797,Z 191,A -78.1825,B 1.0091,C 0.2085,E1 1.0431,E2 531.0299} C_DIS
LIN {X 1.4759,Y -135.7797,Z 191,A -78.1828,B 1.0091,C 0.2085,E1 1.0431,E2 531.0301} C_DIS
Enddeposition()
LIN {X 0.9736,Y -136.6803,Z 191,A -77.9615,B 0.9802,C 0.2065,E1 1.0147,E2 530.7802} C_DIS
Startdeposition()
$VEL.CP = VEL_PRINT
LIN {X 6.5516,Y -136.5279,Z 191,A -75.1528,B 0.9808,C 0.2038,E1 1.0228,E2 527.9025} C_DIS
LIN {X 9.6704,Y -136.3424,Z 191,A -72.9913,B 0.9815,C 0.2003,E1 1.0293,E2 525.6163} C_DIS
LIN {X 16.3992,Y -135.6974,Z 191,A -70.3005,B 0.9818,C 0.1986,E1 1.0367,E2 522.9447} C_DIS
LIN {X 22.9052,Y -134.7522,Z 191,A -68.4101,B 0.9818,C 0.1992,E1 1.0417,E2 521.1786} C_DIS
LIN {X 26.6945,Y -134.0536,Z 191,A -66.9608,B 0.9819,C 0.1983,E1 1.0456,E2 519.7523} C_DIS
LIN {X 30.0201,Y -133.3477,Z 191,A -65.5311,B 0.9822,C 0.1968,E1 1.0496,E2 518.321} C_DIS
LIN {X 33.2989,Y -132.5666,Z 191,A -64.2645,B 0.9824,C 0.1959,E1 1.053,E2 517.0745} C_DIS
LIN {X 36.799,Y -131.6375,Z 191,A -62.9597,B 0.9826,C 0.195,E1 1.0565,E2 515.7994} C_DIS
LIN {X 39.7174,Y -130.7869,Z 191,A -61.6423,B 0.9829,C 0.1933,E1 1.0601,E2 514.4749} C_DIS
LIN {X 45.1799,Y -129.0021,Z 191,A -59.2511,B 0.9835,C 0.1903,E1 1.0664,E2 512.0846} C_DIS
LIN {X 49.0954,Y -127.5634,Z 191,A -57.3764,B 0.984,C 0.1875,E1 1.0714,E2 510.1906} C_DIS
LIN {X 52.5293,Y -126.1874,Z 191,A -55.8888,B 0.9844,C 0.1855,E1 1.0753,E2 508.711} C_DIS
LIN {X 56.2331,Y -124.5817,Z 191,A -54.6828,B 0.9844,C 0.185,E1 1.0782,E2 507.5736} C_DIS
LIN {X 60.0713,Y -122.777,Z 191,A -53.031,B 0.9849,C 0.1828,E1 1.0824,E2 505.9385} C_DIS
LIN {X 62.9664,Y -121.3186,Z 191,A -51.7184,B 0.9853,C 0.1809,E1 1.0856,E2 504.6316} C_DIS
LIN {X 67.052,Y -119.1098,Z 191,A -49.4924,B 0.9861,C 0.1764,E1 1.0912,E2 502.3642} C_DIS
LIN {X 71.1071,Y -116.7343,Z 191,A -47.9734,B 0.9863,C 0.175,E1 1.0947,E2 500.9082} C_DIS
LIN {X 75.6371,Y -113.8518,Z 191,A -45.8154,B 0.987,C 0.1714,E1 1.0998,E2 498.7618} C_DIS
LIN {X 78.5041,Y -111.8936,Z 191,A -44.5964,B 0.9872,C 0.1697,E1 1.1025,E2 497.5753} C_DIS
LIN {X 82.6949,Y -108.834,Z 191,A -42.6809,B 0.9877,C 0.1668,E1 1.1068,E2 495.6949} C_DIS
LIN {X 86.3156,Y -105.9848,Z 191,A -41.112,B 0.9881,C 0.1647,E1 1.1101,E2 494.1757} C_DIS
LIN {X 89.8261,Y -103.0261,Z 191,A -39.0801,B 0.9888,C 0.1602,E1 1.1145,E2 492.1273} C_DIS
LIN {X 93.6599,Y -99.5538,Z 191,A -37.2419,B 0.9893,C 0.1573,E1 1.1182,E2 490.3339} C_DIS
LIN {X 96.8279,Y -96.4754,Z 191,A -35.6197,B 0.9898,C 0.1544,E1 1.1213,E2 488.7423} C_DIS
LIN {X 100.336,Y -92.8213,Z 191,A -33.3463,B 0.9906,C 0.1489,E1 1.1257,E2 486.4462} C_DIS
LIN {X 103.1248,Y -89.7129,Z 191,A -32.1238,B 0.9908,C 0.1476,E1 1.1279,E2 485.2963} C_DIS
LIN {X 105.9949,Y -86.3032,Z 191,A -30.4733,B 0.9913,C 0.1444,E1 1.1308,E2 483.6746} C_DIS
LIN {X 110.2659,Y -80.7748,Z 191,A -27.8883,B 0.992,C 0.1393,E1 1.1351,E2 481.1351} C_DIS
LIN {X 112.0136,Y -78.3336,Z 191,A -26.7113,B 0.9924,C 0.1366,E1 1.137,E2 479.9684} C_DIS
LIN {X 114.7488,Y -74.2688,Z 191,A -24.8939,B 0.9929,C 0.1328,E1 1.1397,E2 478.182} C_DIS
LIN {X 118.0452,Y -68.9099,Z 191,A -22.4772,B 0.9936,C 0.1274,E1 1.1432,E2 475.7937} C_DIS
LIN {X 120.2912,Y -64.9091,Z 191,A -20.6952,B 0.9941,C 0.1233,E1 1.1456,E2 474.0296} C_DIS
LIN {X 122.264,Y -61.1111,Z 191,A -19.1732,B 0.9945,C 0.1201,E1 1.1474,E2 472.5434} C_DIS
LIN {X 124.0073,Y -57.487,Z 191,A -17.8013,B 0.9948,C 0.1174,E1 1.149,E2 471.2129} C_DIS
LIN {X 125.2919,Y -54.6321,Z 191,A -16.1693,B 0.9954,C 0.1123,E1 1.1509,E2 469.5366} C_DIS
LIN {X 127.0834,Y -50.3296,Z 191,A -14.7868,B 0.9956,C 0.1102,E1 1.1523,E2 468.2303} C_DIS
LIN {X 128.2749,Y -47.2095,Z 191,A -12.8556,B 0.9964,C 0.1036,E1 1.1542,E2 466.2261} C_DIS
LIN {X 130.4479,Y -40.8237,Z 191,A -11.0713,B 0.9966,C 0.1016,E1 1.1556,E2 464.5809} C_DIS
LIN {X 131.565,Y -37.0583,Z 191,A -9.7476,B 0.9968,C 0.0989,E1 1.1566,E2 463.2992} C_DIS
LIN {X 132.4501,Y -33.7581,Z 191,A -8.4589,B 0.9971,C 0.0957,E1 1.1575,E2 462.0286} C_DIS
LIN {X 133.1588,Y -30.8471,Z 191,A -7.2911,B 0.9974,C 0.0928,E1 1.1582,E2 460.8717} C_DIS
LIN {X 133.9523,Y -27.1921,Z 191,A -5.9516,B 0.9977,C 0.0897,E1 1.159,E2 459.5614} C_DIS
LIN {X 134.7442,Y -22.9533,Z 191,A -4.4068,B 0.998,C 0.0861,E1 1.1597,E2 458.0503} C_DIS
LIN {X 135.2805,Y -19.5421,Z 191,A -3.0243,B 0.9983,C 0.0825,E1 1.1603,E2 456.6754} C_DIS
LIN {X 136.2712,Y -10.6456,Z 191,A 0.3342,B 0.999,C 0.0742,E1 1.1612,E2 453.3665} C_DIS
LIN {X 136.6641,Y -2.3737,Z 191,A 3.4821,B 0.9995,C 0.0662,E1 1.1615,E2 450.2587} C_DIS
LIN {X 136.6821,Y 0.9749,Z 191,A 4.8664,B 0.9998,C 0.0624,E1 1.1615,E2 448.8762} C_DIS
LIN {X 136.5876,Y 5.1544,Z 191,A 5.7826,B 0.9998,C 0.062,E1 1.1615,E2 448.0669} C_DIS
LIN {X 136.3565,Y 9.4764,Z 191,A 7.8361,B 1.0002,C 0.0556,E1 1.1611,E2 445.9819} C_DIS
LIN {X 136.0968,Y 12.6681,Z 191,A 9.3637,B 1.0004,C 0.0509,E1 1.1607,E2 444.4298} C_DIS
LIN {X 135.4915,Y 18.0218,Z 191,A 10.7799,B 1.0005,C 0.0491,E1 1.1602,E2 443.1203} C_DIS
LIN {X 134.9067,Y 21.9797,Z 191,A 12.2861,B 1.0007,C 0.0454,E1 1.1596,E2 441.635} C_DIS
LIN {X 134.1237,Y 26.3427,Z 191,A 13.967,B 1.0009,C 0.0412,E1 1.1587,E2 439.9757} C_DIS
LIN {X 133.2582,Y 30.4117,Z 191,A 15.38,B 1.0009,C 0.0381,E1 1.1579,E2 438.6035} C_DIS
LIN {X 132.5232,Y 33.4701,Z 191,A 16.4536,B 1.0011,C 0.0358,E1 1.1572,E2 437.5599} C_DIS
LIN {X 131.6836,Y 36.6341,Z 191,A 17.7383,B 1.0011,C 0.0325,E1 1.1562,E2 436.2856} C_DIS
LIN {X 130.7349,Y 39.8872,Z 191,A 19.0196,B 1.0013,C 0.0294,E1 1.1552,E2 435.021} C_DIS
LIN {X 129.7045,Y 43.12,Z 191,A 20.1721,B 1.0013,C 0.027,E1 1.1543,E2 433.9015} C_DIS
LIN {X 128.4062,Y 46.8475,Z 191,A 22.3792,B 1.0015,C 0.0197,E1 1.1521,E2 431.6252} C_DIS
LIN {X 126.3175,Y 52.2177,Z 191,A 23.7445,B 1.0015,C 0.0187,E1 1.1508,E2 430.389} C_DIS
LIN {X 123.6787,Y 58.1959,Z 191,A 26.3922,B 1.0017,C 0.012,E1 1.1478,E2 427.7518} C_DIS
LIN {X 122.0468,Y 61.5418,Z 191,A 27.7138,B 1.0017,C 0.0091,E1 1.1462,E2 426.4589} C_DIS
LIN {X 120.2732,Y 64.9427,Z 191,A 29.1694,B 1.0017,C 0.0058,E1 1.1443,E2 425.0213} C_DIS
LIN {X 118.693,Y 67.787,Z 191,A 30.634,B 1.0017,C 0.0018,E1 1.1422,E2 423.5442} C_DIS
LIN {X 116.7378,Y 71.1026,Z 191,A 31.8403,B 1.0017,C -0.0002,E1 1.1406,E2 422.3869} C_DIS
LIN {X 112.9976,Y 76.9075,Z 191,A 34.4043,B 1.0017,C -0.0057,E1 1.1367,E2 419.862} C_DIS
LIN {X 110.4008,Y 80.5912,Z 191,A 36.1047,B 1.0017,C -0.0093,E1 1.1339,E2 418.1837} C_DIS
LIN {X 107.6848,Y 84.1855,Z 191,A 37.7871,B 1.0017,C -0.0128,E1 1.1311,E2 416.5256} C_DIS
LIN {X 104.8678,Y 87.6693,Z 191,A 39.4443,B 1.0016,C -0.0162,E1 1.1282,E2 414.8942} C_DIS
LIN {X 101.9444,Y 91.0521,Z 191,A 41.1326,B 1.0016,C -0.0196,E1 1.1251,E2 413.2276} C_DIS
LIN {X 98.8411,Y 94.4115,Z 191,A 42.8428,B 1.0015,C -0.0229,E1 1.1219,E2 411.5414} C_DIS
LIN {X 95.5737,Y 97.718,Z 191,A 44.6066,B 1.0014,C -0.0263,E1 1.1184,E2 409.7991} C_DIS
LIN {X 92.2386,Y 100.8725,Z 191,A 46.3225,B 1.0013,C -0.0295,E1 1.1149,E2 408.1074} C_DIS
Enddeposition()
END
